// ---- CNC Beckhoff/6 BlockSearch/ReadBsBlockNumber.TcPOU
FUNCTION_BLOCK ReadBsBlockNumber
VAR_INPUT
	nIdxGrp: UDINT;
	bStart: BOOL;
	pDest: POINTER TO DINT;
END_VAR
VAR_OUTPUT
	Busy: BOOL;
	bErr: BOOL;
END_VAR
VAR
	fbRead: ADSREAD;
	bStarted: BOOL;
END_VAR

IF bStarted = FALSE THEN
   IF bStart = TRUE THEN
      bStarted := TRUE;
      bErr := FALSE;
      Busy := TRUE;
   END_IF
END_IF

IF bStarted THEN
   (* raising edge of Timer triggers read request *)
   fbRead( NetID := '', Port := 553, IdxGrp := nIdxGrp, IdxOffs := 16#00000077,
         LEN := 4, DestAddr := pDest, READ := bStarted, TMOUT := T#1s);
   IF NOT fbRead.Busy THEN
      (* There was an error in the execution of the read request *)
      IF fbRead.Err THEN
         bErr := TRUE;
      END_IF
      fbRead(READ := FALSE);    (* reset because of edge detection in FB ADSREAD *)
      bStarted := FALSE;
      Busy := FALSE;
   END_IF
END_IF

END_FUNCTION_BLOCK

// ---- CNC Beckhoff/6 BlockSearch/WriteBsBlockCount.TcPOU
FUNCTION_BLOCK WriteBsBlockCount
VAR_INPUT
	nIdxGrp: UDINT;
	bStart: BOOL;
	nBlockCount: DINT;
END_VAR
VAR_OUTPUT
	Busy: BOOL;
	bErr: BOOL;
END_VAR
VAR
	fbWrite: ADSWRITE;
	bStarted: BOOL;
END_VAR

IF bStarted = FALSE THEN
   IF bStart = TRUE THEN
      bStarted := TRUE;
      bErr := FALSE;
      Busy := TRUE;
   END_IF
END_IF

IF bStarted THEN
   (* raising edge of Timer triggers write request *)
   fbWrite( NetID := '', Port := 553, IdxGrp := nIdxGrp, IdxOffs := 16#0000005E,
         LEN := 4, SrcAddr := ADR(nBlockCount), WRITE := bStarted, TMOUT := T#1s);
   IF NOT fbWrite.Busy THEN
      (* There was an error in the execution of the write request *)
      IF fbWrite.Err THEN
         bErr := TRUE;
      END_IF
      fbWrite(WRITE := FALSE);    (* reset because of edge detection in FB ADSWRITE *)
      bStarted := FALSE;
      Busy := FALSE;
   END_IF
END_IF

END_FUNCTION_BLOCK

// ---- CNC Beckhoff/6 BlockSearch/ReadBlockCount.TcPOU
FUNCTION_BLOCK ReadBlockCount
VAR_INPUT
	nIdxGrp: UDINT;
	bStart: BOOL;
	pDest: POINTER TO DINT;
END_VAR
VAR_OUTPUT
	Busy: BOOL;
	bErr: BOOL;
END_VAR
VAR
	fbRead: ADSREAD;
	bStarted: BOOL;
END_VAR

IF bStarted = FALSE THEN
   IF bStart = TRUE THEN
      bStarted := TRUE;
      bErr := FALSE;
      Busy := TRUE;
   END_IF
END_IF

IF bStarted THEN
   (* raising edge of Timer triggers read request *)
   fbRead( NetID := '', Port := 553, IdxGrp := nIdxGrp, IdxOffs := 16#0000000D,
         LEN := 4, DestAddr := pDest, READ := bStarted, TMOUT := T#1s);
   IF NOT fbRead.Busy THEN
      (* There was an error in the execution of the read request *)
      IF fbRead.Err THEN
         bErr := TRUE;
      END_IF
      fbRead(READ := FALSE);    (* reset because of edge detection in FB ADSREAD *)
      bStarted := FALSE;
      Busy := FALSE;
   END_IF
END_IF

END_FUNCTION_BLOCK

// ---- CNC Beckhoff/6 BlockSearch/ReadBsBlockCount.TcPOU
FUNCTION_BLOCK ReadBsBlockCount
VAR_INPUT
	nIdxGrp: UDINT;
	bStart: BOOL;
	pDest: POINTER TO DINT;
END_VAR
VAR_OUTPUT
	Busy: BOOL;
	bErr: BOOL;
END_VAR
VAR
	fbRead: ADSREAD;
	bStarted: BOOL;
END_VAR

IF bStarted = FALSE THEN
   IF bStart = TRUE THEN
      bStarted := TRUE;
      bErr := FALSE;
      Busy := TRUE;
   END_IF
END_IF

IF bStarted THEN
   (* raising edge of Timer triggers read request *)
   fbRead( NetID := '', Port := 553, IdxGrp := nIdxGrp, IdxOffs := 16#00000076,
         LEN := 4, DestAddr := pDest, READ := bStarted, TMOUT := T#1s);
   IF NOT fbRead.Busy THEN
      (* There was an error in the execution of the read request *)
      IF fbRead.Err THEN
         bErr := TRUE;
      END_IF
      fbRead(READ := FALSE);    (* reset because of edge detection in FB ADSREAD *)
      bStarted := FALSE;
      Busy := FALSE;
   END_IF
END_IF

END_FUNCTION_BLOCK

// ---- CNC Beckhoff/6 BlockSearch/WriteBsPass.TcPOU
FUNCTION_BLOCK WriteBsPass
VAR_INPUT
	nIdxGrp: UDINT;
	bStart: BOOL;
	nPass: DINT;
END_VAR
VAR_OUTPUT
	Busy: BOOL;
	bErr: BOOL;
END_VAR
VAR
	fbWrite: ADSWRITE;
	bStarted: BOOL;
END_VAR

IF bStarted = FALSE THEN
   IF bStart = TRUE THEN
      bStarted := TRUE;
      bErr := FALSE;
      Busy := TRUE;
   END_IF
END_IF

IF bStarted THEN
   (* raising edge of Timer triggers write request *)
   fbWrite( NetID := '', Port := 553, IdxGrp := nIdxGrp, IdxOffs := 16#00000060,
         LEN := 4, SrcAddr := ADR(nPass), WRITE := bStarted, TMOUT := T#1s);
   IF NOT fbWrite.Busy THEN
      (* There was an error in the execution of the write request *)
      IF fbWrite.Err THEN
         bErr := TRUE;
      END_IF
      fbWrite(WRITE := FALSE);    (* reset because of edge detection in FB ADSWRITE *)
      bStarted := FALSE;
      Busy := FALSE;
   END_IF
END_IF

END_FUNCTION_BLOCK

// ---- CNC Beckhoff/6 BlockSearch/ReadBsPass.TcPOU
FUNCTION_BLOCK ReadBsPass
VAR_INPUT
	nIdxGrp: UDINT;
	bStart: BOOL;
	pDest: POINTER TO DINT;
END_VAR
VAR_OUTPUT
	Busy: BOOL;
	bErr: BOOL;
END_VAR
VAR
	fbRead: ADSREAD;
	bStarted: BOOL;
END_VAR

IF bStarted = FALSE THEN
   IF bStart = TRUE THEN
      bStarted := TRUE;
      bErr := FALSE;
      Busy := TRUE;
   END_IF
END_IF

IF bStarted THEN
   (* raising edge of Timer triggers read request *)
   fbRead( NetID := '', Port := 553, IdxGrp := nIdxGrp, IdxOffs := 16#00000078,
         LEN := 4, DestAddr := pDest, READ := bStarted, TMOUT := T#1s);
   IF NOT fbRead.Busy THEN
      (* There was an error in the execution of the read request *)
      IF fbRead.Err THEN
         bErr := TRUE;
      END_IF
      fbRead(READ := FALSE);    (* reset because of edge detection in FB ADSREAD *)
      bStarted := FALSE;
      Busy := FALSE;
   END_IF
END_IF

END_FUNCTION_BLOCK

// ---- CNC Beckhoff/2 OperationMode/ModeManual/HLI3_ManualModeHandler.TcPOU
FUNCTION_BLOCK HLI3_ManualModeHandler
VAR_INPUT
	stManualModeParameter: ST_ManualModeParameter;
	stManualModeControlElements: ST_ManualModeControlElements;
	bReset: BOOL;
END_VAR
VAR_OUTPUT
	bInManualMode: BOOL;
	arrAxisInG201: ARRAY[0..HLI_KEY_MAXIDX] OF UINT;
	bBusy: BOOL;
	bError: BOOL;
	nErrorId: INT;
END_VAR
VAR_IN_OUT
	stManualModeControlElementState: ST_ManualModeControlElementState;
END_VAR
VAR
	nState: INT;
	pString: POINTER TO STRING;
	pUnit: POINTER TO MC_CONTROL_MCM_MODE_STATE_UNIT;
	pCommand: POINTER TO HLI_PROC_TRANS_TO_MODE_STATE;
	pKey: POINTER TO MC_CONTROL_HB_KEY_UNIT;
	pIncr: POINTER TO MC_CONTROL_HB_TIP_PARAM_UNIT;
	stManualModeParameterOld: ST_ManualModeParameter;
	incOld: UINT;
	nManualTypOld: UINT;
	i: INT;
	bManual: BOOL;
	/// FBs for manual mode 
	ManualActivation: HLI3_ManualActivation;
	ManualExecution: ARRAY[0..HLI_KEY_MAXIDX] OF HLI3_ManualExecution;
	ManualExecutionRapidMode: ARRAY[0..HLI_KEY_MAXIDX] OF HLI3_ManualExecutionRapidMode;
	ActChannelModeOld: UDINT;
	TON_TimeOut: TON;
	nChan: INT;
	j: INT;
	strInitParameterOld: STRING;
	bInJoystickMode: BOOL;
	nHliAxisIdx: INT;
	nControlUnit: INT;
	arrAxisInJoystickMode: ARRAY[0..HLI_KEY_MAXIDX] OF UINT;
	n: INT;
	bInit: BOOL;
END_VAR
VAR CONSTANT
	ErrID_1: INT := 1;
END_VAR

(* ========================================================= 	*)
(*     FB: HLI3_ManualModeHandler                           	*)
(* --------------------------------------------------------- 	*)
(*   Desc: Switch to Manual Mode and parametrize             	*)
(*   Author: MK / TV  /MiB                                      *)
(*   Date: 18.07.2002                                        	*)
(*   Last: 18.11.2015                                        	*)
(*   Rev.: 6.4	                                              	*)
(* ========================================================= 	*)

nChan := stManualModeParameter.stChannelParameter.nChanIdx;
IF (NOT HLI3_CheckChannelValid(nChannel := nChan) OR nChan = -1 )  THEN
	RETURN;
END_IF

IF NOT bInit THEN  
	gpCh[nChan]^.hb_mc_control.activation.enable_w := TRUE;
	FOR j := 0 TO HLI_HW_MAXIDX DO
		gpCh[nChan]^.hb_mc_control.handwheel_incs[j].enable_w  := TRUE;
	END_FOR
	bInit := TRUE;
END_IF	

IF 	CNCSystem.Channel[nChan].ActMode <> HLI_IMCM_MANUAL_MODE AND
	CNCSystem.Channel[nChan].ActMode <> HLI_IMCM_AUTOMATIC_MODE   AND
	CNCSystem.Channel[nChan].ActMode <> HLI_IMCM_MDI_MODE THEN
		strInitParameterOld := '';
		bBusy := FALSE;
		nState := 0;
	RETURN; (* A b b r u c h *)
ELSE
	bManual := TRUE;
END_IF

IF  CNCSystem.Channel[nChan].ActMode <> HLI_IMCM_MANUAL_MODE THEN
	strInitParameterOld := '';
END_IF

(* Clear all request from the HMI *)
IF gpCh[nChan]^.hb_mc_control.key[0].request_semaphor_rw THEN
	gpCh[nChan]^.hb_mc_control.key[0].request_semaphor_rw := FALSE;
END_IF

IF gpCh[nChan]^.hb_mc_control.activation.request_semaphor_rw THEN
	gpCh[nChan]^.hb_mc_control.activation.request_semaphor_rw := FALSE;
END_IF

IF gpCh[nChan]^.hb_mc_control.tip_parameter.request_semaphor_rw THEN
	gpCh[nChan]^.hb_mc_control.tip_parameter.request_semaphor_rw := FALSE;
END_IF

IF gpCh[nChan]^.hb_mc_control.jog_parameter.request_semaphor_rw THEN
	gpCh[nChan]^.hb_mc_control.jog_parameter.request_semaphor_rw := FALSE;
END_IF

bBusy := TRUE;

IF bReset THEN		
	bError := FALSE;
	nErrorID := 0;
	bInManualMode := FALSE;
END_IF


IF stManualModeParameter.stChannelParameter.eManualType = E_CNC_ManualType.JoystickMode THEN

	bInJoystickMode := TRUE;
	
	arrAxisInJoystickMode := HLI3_LogicalAxisInManualMode(nCHan);
	
	PRG_AnalogJoystick(	nLogAxisNr:= stManualModeParameter.stAxisParameter.stControlUnit[0].nLogAxisNr,
								Analog_Value:= stManualModeControlElements.stControlJoystickValue[0],
								AnalogValueMin:= stManualModeParameter.stJoystickParameter.AnalogValueMin,
								AnalogValueMax:= stManualModeParameter.stJoystickParameter.AnalogValueMax,
								AnalogValueZeroDeadBand:= stManualModeParameter.stJoystickParameter.AnalogValueZeroDeadBand,
								bKeyPos:= stManualModeControlElements.stControlKeys[0].bKeyPos,
								bKeyNeg:= stManualModeControlElements.stControlKeys[0].bKeyNeg);

	PRG_AnalogJoystick(	nLogAxisNr:= stManualModeParameter.stAxisParameter.stControlUnit[1].nLogAxisNr,
								Analog_Value:= stManualModeControlElements.stControlJoystickValue[1],
								AnalogValueMin:= stManualModeParameter.stJoystickParameter.AnalogValueMin,
								AnalogValueMax:= stManualModeParameter.stJoystickParameter.AnalogValueMax,
								AnalogValueZeroDeadBand:= stManualModeParameter.stJoystickParameter.AnalogValueZeroDeadBand,
								bKeyPos:= stManualModeControlElements.stControlKeys[1].bKeyPos,
								bKeyNeg:= stManualModeControlElements.stControlKeys[1].bKeyNeg);

	PRG_AnalogJoystick(	nLogAxisNr:= stManualModeParameter.stAxisParameter.stControlUnit[2].nLogAxisNr,
								Analog_Value:= stManualModeControlElements.stControlJoystickValue[2],
								AnalogValueMin:= stManualModeParameter.stJoystickParameter.AnalogValueMin,
								AnalogValueMax:= stManualModeParameter.stJoystickParameter.AnalogValueMax,
								AnalogValueZeroDeadBand:= stManualModeParameter.stJoystickParameter.AnalogValueZeroDeadBand,
								bKeyPos:= stManualModeControlElements.stControlKeys[2].bKeyPos,
								bKeyNeg:= stManualModeControlElements.stControlKeys[2].bKeyNeg);

	PRG_AnalogJoystick(	nLogAxisNr:= stManualModeParameter.stAxisParameter.stControlUnit[3].nLogAxisNr,
								Analog_Value:= stManualModeControlElements.stControlJoystickValue[3],
								AnalogValueMin:= stManualModeParameter.stJoystickParameter.AnalogValueMin,
								AnalogValueMax:= stManualModeParameter.stJoystickParameter.AnalogValueMax,
								AnalogValueZeroDeadBand:= stManualModeParameter.stJoystickParameter.AnalogValueZeroDeadBand,
								bKeyPos:= stManualModeControlElements.stControlKeys[3].bKeyPos,
								bKeyNeg:= stManualModeControlElements.stControlKeys[3].bKeyNeg);

	PRG_AnalogJoystick(	nLogAxisNr:= stManualModeParameter.stAxisParameter.stControlUnit[4].nLogAxisNr,
								Analog_Value:= stManualModeControlElements.stControlJoystickValue[4],
								AnalogValueMin:= stManualModeParameter.stJoystickParameter.AnalogValueMin,
								AnalogValueMax:= stManualModeParameter.stJoystickParameter.AnalogValueMax,
								AnalogValueZeroDeadBand:= stManualModeParameter.stJoystickParameter.AnalogValueZeroDeadBand,
								bKeyPos:= stManualModeControlElements.stControlKeys[4].bKeyPos,
								bKeyNeg:= stManualModeControlElements.stControlKeys[4].bKeyNeg);

ELSE
	(* Achsoverride wieder auf 100 % setzen *)
	IF bInJoystickMode THEN 
		nHliAxisIdx := -1;
		FOR j := 0 TO UINT_TO_INT(SIZEOF(arrAxisInJoystickMode)) DO
			FOR i := 0 TO UDINT_TO_INT(gNrAx-1) DO
				IF (gpAX[i]^.head.log_ax_nr_r = arrAxisInJoystickMode[j]) THEN
					nHliAxisIdx := i;	
					IF (nHliAxisIdx <> -1) THEN 
						HLI3_SetAxisOverride(nHliAxisIdx := nHliAxisIdx, nOverride := 1000);
						nHliAxisIdx := -1;
						arrAxisInJoystickMode[j] := 0;
					END_IF								
				END_IF
			END_FOR			
		END_FOR
		bInJoystickMode := FALSE;
	END_IF
END_IF

(******** Parallelinterpolation mit G201 *************************************)
IF CNCSystem.Channel[nChan].ActMode = HLI_IMCM_AUTOMATIC_MODE OR CNCSystem.Channel[nChan].ActMode = HLI_IMCM_MDI_MODE THEN
	arrAxisInG201 := HLI3_LogicalAxisInManualMode(nCHan);
	FOR j := 0 TO HLI_KEY_MAXIDX DO
		stManualModeParameter.stAxisParameter.stControlUnit[j].nLogAxisNr := arrAxisInG201[j];
	END_FOR
ELSE
	FOR j := 0 TO HLI_KEY_MAXIDX DO
		arrAxisInG201[j] := 0;
	END_FOR
END_IF
(* **************************************************************************** *)

IF NOT gpCh[nChan]^.bahn_state.g201_active_r THEN
	IF CNCSystem.Channel[nChan].ActMode = HLI_IMCM_AUTOMATIC_MODE OR CNCSystem.Channel[nChan].ActMode = HLI_IMCM_MDI_MODE THEN
		nState := 0; 
	END_IF
END_IF

CASE nState OF


	0: (* IDLE *)
		bBusy := FALSE;
		bInManualMode := FALSE;


		IF (CNCSystem.Channel[nChan].ActMode = HLI_IMCM_MANUAL_MODE AND
    		stManualModeParameter.stChannelParameter.eManualType <> E_CNC_ManualType.NoManualMode AND
    		CNCSystem.Channel[nChan].ActState = HLI_IMCM_PROCESS_ACTIVE) OR  (* Manual Mode *)
   			((arrAxisinG201[0] <> 0)    (* mindestens eine Achse in G201 *) AND
    		((CNCSystem.Channel[nChan].ActState = HLI_IMCM_PROCESS_ACTIVE) OR
     		(CNCSystem.Channel[nChan].ActState = HLI_IMCM_PROCESS_HOLD))) (* Channel is active *)
		THEN			
			bError 		:= FALSE;
			nErrorID 	:= 0;

			stManualModeParameterOld     := stManualModeParameter;
			ActChannelModeOld   		:= cncsystem.Channel[nChan].ActMode;			
			i:= 0;
			nState := 10;

		END_IF

	10:		// Restore Manual State										
			FOR j := 0 TO HLI_KEY_MAXIDX DO
				IF (stManualModeControlElementState.stKeyUnit[j].nChan = nChan) THEN
					stManualModeControlElementState.stKeyUnit[j].nChan := -1;
					stManualModeControlElementState.stKeyUnit[j].nLogAxisId := 0;
					stManualModeControlElementState.stKeyUnit[j].nInputParameterIdx := -1;
				END_IF													
			END_FOR
			
			FOR j := 0 TO HLI_HW_MAXIDX DO
				IF (stManualModeControlElementState.stHWUnit[j].nChan = nChan) THEN
					stManualModeControlElementState.stHWUnit[j].nChan := -1;
					stManualModeControlElementState.stHWUnit[j].nLogAxisId := 0;
					stManualModeControlElementState.stHWUnit[j].nInputParameterIdx := -1;
				END_IF													
			END_FOR
			(*
			FOR j := 0 TO HLI_CH_AX_MAXIDX DO
				IF gpCh[nChan]^.bahn_state.coord_r[j].hb_display_r.control_element <> 0 THEN
					IF gpCh[nChan]^.bahn_state.coord_r[j].hb_display_r.operation_mode = 1 THEN  
						stManualModeControlElementState.stHWUnit[gpCh[nChan]^.bahn_state.coord_r[j].hb_display_r.control_element-1].nLogAxisId := gpCh[nChan]^.bahn_state.coord_r[j].log_achs_nr_r;
 						stManualModeControlElementState.stHWUnit[gpCh[nChan]^.bahn_state.coord_r[j].hb_display_r.control_element-1].nChan := nChan;
					ELSE
						stManualModeControlElementState.stKeyUnit[gpCh[nChan]^.bahn_state.coord_r[j].hb_display_r.control_element-1].nLogAxisId := gpCh[nChan]^.bahn_state.coord_r[j].log_achs_nr_r;
 						stManualModeControlElementState.stKeyUnit[gpCh[nChan]^.bahn_state.coord_r[j].hb_display_r.control_element-1].nChan := nChan;
					END_IF
				END_IF 
			END_FOR
*)	
			n:= 0;		
			nState := 20;						
			
20: 	// Deactivation 
		IF (n <= HLI_CH_AX_MAXIDX) THEN
			IF gpCh[nChan]^.bahn_state.coord_r[n].hb_display_r.control_element <> 0 THEN 
				IF NOT gpCh[nChan]^.hb_mc_control.activation.command_semaphor_rw THEN		
						gpCh[nChan]^.hb_mc_control.activation.command_w.log_achs_nr := gpCh[nChan]^.bahn_state.coord_r[n].log_achs_nr_r;
						gpCh[nChan]^.hb_mc_control.activation.command_w.control_element := 0;
						gpCh[nChan]^.hb_mc_control.activation.command_w.operation_mode := 0;
						
						IF (gpCh[nChan]^.bahn_state.coord_r[n].hb_display_r.operation_mode = 1) THEN
							stManualModeControlElementState.stHWUnit[gpCh[nChan]^.bahn_state.coord_r[n].hb_display_r.control_element-1].nChan := -1;
							stManualModeControlElementState.stHWUnit[gpCh[nChan]^.bahn_state.coord_r[n].hb_display_r.control_element-1].nLogAxisId :=0;
							stManualModeControlElementState.stHWUnit[gpCh[nChan]^.bahn_state.coord_r[n].hb_display_r.control_element-1].nInputParameterIdx := -1;	
						ELSE
							stManualModeControlElementState.stKeyUnit[gpCh[nChan]^.bahn_state.coord_r[n].hb_display_r.control_element-1].nChan := -1;
							stManualModeControlElementState.stKeyUnit[gpCh[nChan]^.bahn_state.coord_r[n].hb_display_r.control_element-1].nLogAxisId :=0;
							stManualModeControlElementState.stKeyUnit[gpCh[nChan]^.bahn_state.coord_r[n].hb_display_r.control_element-1].nInputParameterIdx := -1;						
						END_IF
						gpCh[nChan]^.hb_mc_control.activation.command_semaphor_rw := TRUE;
						nState := 21;					
				END_IF
			ELSE
				n := n + 1;
			END_IF				
		END_IF

		IF n >HLI_CH_AX_MAXIDX THEN
			nState := 26;
		END_IF
21: 
		IF 	NOT gpCh[nChan]^.hb_mc_control.activation.command_semaphor_rw THEN						
			n := n+1;
			nState := 20;
		END_IF
		
		IF n > HLI_CH_AX_MAXIDX THEN
			nState := 26;
		END_IF			
			 					
		(* Activation of an manual mode string, eg. TRAFO ON or ECS ON *)
26:     IF 	(stManualModeParameter.stChannelParameter.strInitParameter  <> '' AND
			stManualModeParameter.stChannelParameter.strInitParameter <> strInitParameterOld AND
			CNCSystem.Channel[nChan].ActMode = HLI_IMCM_MANUAL_MODE) THEN
			gpCh[nCHan]^.channel_mc_control.mode_and_state.command_w.to_mode := HLI_IMCM_MANUAL_MODE ;
			gpCh[nCHan]^.channel_mc_control.mode_and_state.command_w.to_state := HLI_IMCM_PROCESS_SELECTED;
			gpCh[nCHan]^.channel_mc_control.mode_and_state.command_w.channel_number := INT_TO_UDINT(nChan+1);
			pString := ADR(gpCh[nCHan]^.channel_mc_control.mode_and_state.command_w.parameter);
			pString^ := '';
			gpCh[nChan]^.channel_mc_control.mode_and_state.command_semaphor_rw := TRUE;
			TON_TimeOut(in:= FALSE);
			nState := 27;
		ELSE
			i := 0;
			nState := 30;
		END_IF


27:		IF (gpCh[nCHan]^.channel_mc_control.mode_and_state.command_semaphor_rw = FALSE) AND 
			CNCSystem.Channel[nChan].ActState = HLI_IMCM_PROCESS_SELECTED 
		THEN
			gpCh[nCHan]^.channel_mc_control.mode_and_state.command_w.to_mode := HLI_IMCM_MANUAL_MODE ;
			gpCh[nCHan]^.channel_mc_control.mode_and_state.command_w.to_state := HLI_IMCM_PROCESS_ACTIVE;
			gpCh[nCHan]^.channel_mc_control.mode_and_state.command_w.channel_number := INT_TO_UDINT(nChan+1);
			pString := ADR(gpCh[nCHan]^.channel_mc_control.mode_and_state.command_w.parameter);
			pString^ := stManualModeParameter.stChannelParameter.strInitParameter;
			gpCh[nCHan]^.channel_mc_control.mode_and_state.command_semaphor_rw := TRUE;		
			TON_TimeOut(in:= FALSE);		
			nState := 28;
		END_IF

		TON_TimeOut(in:=TRUE, PT:=T#5s);
		IF TON_TimeOut.Q THEN
			nState := 99;
		END_IF

28:		IF (gpCh[nCHan]^.channel_mc_control.mode_and_state.command_semaphor_rw = FALSE)  AND
			CNCSystem.Channel[nChan].ActState = HLI_IMCM_PROCESS_ACTIVE 
			THEN														
				strInitParameterOld := stManualModeParameter.stChannelParameter.strInitParameter;
				ManualActivation(bExecute := FALSE,stManualModeControlElementState:= stManualModeControlElementState);
				i := 0;
				IF (gpCh[nChan]^.bahn_state.g200_active_r) THEN	
					nState := 30;
				END_IF
						
		END_IF	

		// Abbruch wenn die Betriebsart gewechselt wird 
		IF (CNCSystem.Channel[nChan].ActMode <> HLI_IMCM_MANUAL_MODE) THEN
			nState := 0;
		END_IF	
	
30: 	(* --- activate KeyControlUnits --- *)														
		ManualActivation(bExecute := TRUE,
									nChan 			 := nChan,
									eManualType 	 := stManualModeParameter.stChannelParameter.eManualType,									
									stManualModeControlElementState:= stManualModeControlElementState,
									nInputParameterIdx := i,
									nHBA_Res 		 := stManualModeParameter.stChannelParameter.nHandwheelResolution,
									Inc 		     := stManualModeParameter.stChannelParameter.nInc,
									Speed 			 := stManualModeParameter.stAxisParameter.stControlUnit[i].nSpeed, // geändert alt nControlUnit
									nLogAxisNr 		 := stManualModeParameter.stAxisParameter.stControlUnit[i].nLogAxisNr); // geändert alt nControlUnit
		nState := 35;				
															
35: 	(* waiting for acknowledge *)
		ManualActivation(bExecute := FALSE, stManualModeControlElementState:= stManualModeControlElementState);
		
		IF ManualActivation.bBusy = FALSE THEN
			IF ManualActivation.bError THEN
				nErrorId := ErrID_1;
				nState := 99;
			ELSE
				IF stManualModeParameter.stAxisParameter.stControlUnit[i+1].nLogAxisNr = 0 THEN
					i:=-1; (* reset the array counter *)				
					nState := 40;
				ELSE
					ManualActivation(bExecute := FALSE, stManualModeControlElementState:= stManualModeControlElementState);
					nState := 30;
					i:= i+1;
				END_IF
			END_IF
		END_IF

40: 	(* endlich Handbetrieb *)
		bInManualMode := TRUE;
		
		IF (stManualModeParameter.stChannelParameter.eManualType <> E_CNC_ManualType.Handwheel) THEN
			FOR j := 0 TO HLI_KEY_MAXIDX DO
				IF stManualModeControlElementState.stKeyUnit[j].nChan = nChan AND stManualModeControlElementState.stKeyUnit[j].nLogAxisId <> 0 THEN				
					ManualExecution[j](	nChan := nChan,
									nKeyControlUnit := j,
									bKeyPos := stManualModeControlElements.stControlKeys[stManualModeControlElementState.stKeyUnit[j].nInputParameterIdx].bKeyPos,					// geändert 	nControlUnit
									bKeyNeg := stManualModeControlElements.stControlKeys[stManualModeControlElementState.stKeyUnit[j].nInputParameterIdx].bKeyNeg); (* no timeouts *)
									
					ManualExecutionRapidMode[j](nChan := nChan,
									nKeyControlUnit := j,
									bExecute := stManualModeControlElements.stControlKeys[stManualModeControlElementState.stKeyUnit[j].nInputParameterIdx].bKeyRapid); (* no timeouts *)
				END_IF
			END_FOR			
		ELSE				
			(* Handradincremente werden immer vom ersten Kanal entgegen genommen*)
			FOR j := 0 TO HLI_HW_MAXIDX DO
				IF (stManualModeControlElementState.stHWUnit[j].nChan = nChan AND stManualModeControlElementState.stHWUnit[j].nLogAxisId <>  0)  THEN 
					gpCh[0]^.hb_mc_control.handwheel_incs[j].command_w := stManualModeControlElements.nHandwheelInc[stManualModeControlElementState.stHWUnit[j].nInputParameterIdx];
				END_IF			
			END_FOR
		END_IF

		(* end of manual mode *)
		 IF (bManual = FALSE) OR                                                                                                             
         	MEMCMP(ADR(stManualModeParameter),ADR(stManualModeParameterOld),SIZEOF(stManualModeParameter)-SIZEOF(stManualModeParameter.stChannelParameter.strInitParameter))<>0 OR                                                      
            stManualModeParameter.stChannelParameter.strInitParameter <> stManualModeParameterOld.stChannelParameter.strInitParameter OR                                                          
            cncsystem.Channel[nChan].ActMode <> ActChannelModeOld OR                                       
            (CNCSystem.Channel[nChan].ActMode =  HLI_IMCM_MANUAL_MODE AND CNCSystem.Channel[nChan].ActState <> HLI_IMCM_PROCESS_ACTIVE) OR                                                   
            stManualModeParameter.stChannelParameter.eManualType = E_CNC_ManualType.NoManualMode
            THEN
		
				FOR j := 0 TO HLI_KEY_MAXIDX DO
					IF stManualModeControlElementState.stKeyUnit[j].nChan = nChan THEN
						ManualExecution[j](nChan := nChan,	nKeyControlUnit := j, bKeyPos := FALSE, bKeyNeg := FALSE); (* no timeouts *)		
					END_IF		
				END_FOR
						
				i:=1 (* resets the counter for the following deactivation *);			

				stManualModeParameterOld 	:= stManualModeParameter;
	
				IF cncsystem.Channel[nChan].ActMode <> ActChannelModeOld OR stManualModeParameter.stChannelParameter.eManualType = E_CNC_ManualType.NoManualMode THEN
					ActChannelModeOld := cncsystem.Channel[nChan].ActMode;			
					nState := 0;
				ELSE
					nState := 0; (* evt. wird hier auch eine Verzoegerungszeit benötigt,
										  Fehler 150054 dann nState = 0 *)
					bInManualMode := FALSE;
				END_IF
		END_IF

99: 	(* error handling *)	
		bBusy := FALSE;
		bError := TRUE;
		
		(* end of manual mode *)
			IF NOT gpCh[nCHan]^.channel_mc_control.mode_and_state.command_semaphor_rw AND 
			CNCSystem.Channel[nChan].ActState <>  HLI_IMCM_PROCESS_ERROR
			THEN;
				gpCh[nCHan]^.channel_mc_control.mode_and_state.command_w.to_mode := HLI_IMCM_MANUAL_MODE ;
				gpCh[nCHan]^.channel_mc_control.mode_and_state.command_w.to_state := HLI_IMCM_PROCESS_ERROR;
				gpCh[nCHan]^.channel_mc_control.mode_and_state.command_w.channel_number := INT_TO_UDINT(nChan+1);			
				gpCh[nCHan]^.channel_mc_control.mode_and_state.command_semaphor_rw := TRUE;	
			END_IF
			nState := 0;
		
		(* end of manual mode *)
		IF bManual = FALSE THEN
			bBusy := FALSE;
			nState := 0;
		END_IF

END_CASE

END_FUNCTION_BLOCK

// ---- CNC Beckhoff/2 OperationMode/ModeManual/HLI3_ManualActivation.TcPOU
FUNCTION_BLOCK HLI3_ManualActivation
VAR_INPUT
	bExecute: BOOL;
	/// Number of channel 
	nChan: INT;
	eManualType: E_CNC_ManualType;
	/// Increments -> 0 activates Tip mode 
	Inc: UDINT;
	/// Aufloesung des Achsverfahrwegs bei einer Handradumdrehung Einheit: 0.1um / Handradumdrehung
	nHBA_Res: DINT;
	Speed: UDINT;
	/// axis nr 
	nLogAxisNr: UINT;
	nInputParameterIdx: INT;
END_VAR
VAR_OUTPUT
	bError: BOOL;
	bBusy: BOOL;
END_VAR
VAR_IN_OUT
	stManualModeControlElementState: ST_ManualModeControlElementState;
END_VAR
VAR
	fbRtrigExec: R_TRIG;
	nState: INT;
	pActivation: POINTER TO MC_CONTROL_HB_ACTIVATION_UNIT;
	pJogParameter: POINTER TO MC_CONTROL_HB_JOG_PARAM_UNIT;
	pTipParameter: POINTER TO MC_CONTROL_HB_TIP_PARAM_UNIT;
	pHBHRParameter: POINTER TO MC_CONTROL_HB_HR_PARAM_UNIT;
	j: INT;
	bFreeControlElementFound: BOOL;
END_VAR

(* ========================================================= *)
(*    FUN: HLI_ManualActivation                       		 *)
(* --------------------------------------------------------- *)
(*   Desc:                                                   *)
(*   Author: CL TV MiB                                       *)
(*   Date: 18.11.2005                                        *)
(*   Last: 25.02.2015                                       *)
(*   Rev.: 6.0                                              *)
(* ========================================================= *)

IF NOT HLI3_CheckChannelValid(nChannel := nChan) OR nLogAxisNr = 0 THEN
	RETURN;
END_IF


fbRtrigExec(clk := bExecute);
IF fbRtrigExec.Q THEN
	bBusy := TRUE;
	bError := FALSE;
	nState := 10;
END_IF

CASE nState OF

	0: (* IDLE *)
		bBusy := FALSE;

	10:
		CASE eManualType OF
			E_CNC_ManualType.NoManualMode: 
				nState := 100;

			E_CNC_ManualType.Handwheel:
				nState := 30;

			E_CNC_ManualType.TippMode:
				nState := 40;

			E_CNC_ManualType.JogMode:
				nState := 50;

			E_CNC_ManualType.JoystickMode:
				nState := 40;

			E_CNC_ManualType.DigitalJoystick: 
				nState := 40;

		END_CASE

	30:(* Setze Handrad Parameter *)
		pHBHRParameter := ADR(gpCh[nChan]^.hb_mc_control.hr_parameter);
		IF NOT pHBHRParameter^.command_semaphor_rw THEN
			pHBHRParameter^.enable_w := TRUE;
			pHBHRParameter^.command_w.resolution  := nHBA_Res;
			pHBHRParameter^.command_w.log_achs_nr := nLogAxisNr;
			pHBHRParameter^.command_semaphor_rw := TRUE;
			nState := 100;
		END_IF

	40: (* Setze Parameter für den Tippbetrieb *)
		pTipParameter := ADR(gpCh[nChan]^.hb_mc_control.tip_parameter);
		IF NOT pTipParameter^.command_semaphor_rw THEN
			pTipParameter^.enable_w := TRUE;
			pTipParameter^.command_w.log_achs_nr := nLogAxisNr;
			pTipParameter^.command_w.speed       := Speed;
			pTipParameter^.command_semaphor_rw := TRUE;
			nState := 100;
		END_IF

	50: (* Setze Parameter für den Jogbetrieb *)
		pJogParameter := ADR(gpCh[nChan]^.hb_mc_control.jog_parameter);
		IF NOT pJogParameter^.command_semaphor_rw THEN
			pJogParameter^.enable_w := TRUE;
			pJogParameter^.command_w.log_achs_nr := nLogAxisNr;
			pJogParameter^.command_w.distance    := Inc;
			pJogParameter^.command_w.speed       := Speed;
			pJogParameter^.command_semaphor_rw := TRUE;
			nState := 100;
		END_IF		
		
	100: 	(* Aktivierung der Bedienelementen für den Handbetrieb  *)		
		
		pActivation := ADR(gpCh[nChan]^.hb_mc_control.activation);
		IF NOT pActivation^.command_semaphor_rw THEN 
			bFreeControlElementFound := FALSE;


			IF 	eManualType <> E_CNC_ManualType.Handwheel THEN 	
				FOR j := 0 TO HLI_KEY_MAXIDX DO
					IF stManualModeControlElementState.stKeyUnit[j].nLogAxisId = 0 THEN
							stManualModeControlElementState.stKeyUnit[j].nLogAxisId := nLogAxisNr;
							stManualModeControlElementState.stKeyUnit[j].nChan := nChan;
							stManualModeControlElementState.stKeyUnit[j].nInputParameterIdx := nInputParameterIdx;
							bFreeControlElementFound := TRUE;
						EXIT;
					END_IF 
				END_FOR
			ELSE
				FOR j := 0 TO HLI_HW_MAXIDX DO
					IF stManualModeControlElementState.stHWUnit[j].nLogAxisId = 0 THEN
							stManualModeControlElementState.stHWUnit[j].nLogAxisId := nLogAxisNr;
							stManualModeControlElementState.stHWUnit[j].nChan := nChan;
							stManualModeControlElementState.stHWUnit[j].nInputParameterIdx := nInputParameterIdx;
							bFreeControlElementFound := TRUE;
						EXIT;
					END_IF 
				END_FOR
			END_IF
							
			IF bFreeControlElementFound THEN
				pActivation^.enable_w := TRUE;
				pActivation^.command_w.log_achs_nr := nLogAxisNr;
				pActivation^.command_w.control_element := INT_TO_UINT(j+1);
		
		
				CASE eManualType OF
					E_CNC_ManualType.NoManualMode: 
						pActivation^.command_w.operation_mode := 0; 	(* 0 - No OP_Mode *)
		
					E_CNC_ManualType.Handwheel: 
						pActivation^.command_w.operation_mode := 1; 	(* 1 - Handwheel *)
		
					E_CNC_ManualType.TippMode: 
						pActivation^.command_w.operation_mode := 2; 	(* 2 - Tip Mode continous *)
		
					E_CNC_ManualType.JogMode: 
						pActivation^.command_w.operation_mode := 3; 	(* 3 - Jog Mode (incremental *)
		
					E_CNC_ManualType.JoystickMode: 
						pActivation^.command_w.operation_mode := 2; 	(* 2 - Tip Mode continous, auch für Analog Joystick *)
		
					E_CNC_ManualType.DigitalJoystick: 
						pActivation^.command_w.operation_mode := 2; 	(* 2 - Tip Mode continous, auch für Digital Joystick *)
		
				END_CASE
			
				pActivation^.command_semaphor_rw := TRUE;
				nState := 0;
			ELSE
				bError := TRUE;
				nState := 0;
			END_IF
		END_IF						
END_CASE

END_FUNCTION_BLOCK

// ---- CNC Beckhoff/2 OperationMode/ModeManual/HLI3_ManualExecution.TcPOU
FUNCTION_BLOCK HLI3_ManualExecution
VAR_INPUT
	nChan: INT;
	/// number of the HB_KeyControlUnit 
	nKeyControlUnit: INT;
	/// static signal 
	bKeyPos: BOOL;
	/// static signal 
	bKeyNeg: BOOL;
END_VAR
VAR
	Cmd_Dir: E_HLI_MM_KEYDirection;
	Act_Dir: E_HLI_MM_KEYDirection;
END_VAR

(* ========================================================= *)
(*    FUN: HLI_ManualExecution                    		 		 *)
(* --------------------------------------------------------- *)
(*   Desc:                                                   *)
(*   Author: CL / TV                                         *)
(*   Date: 24.07.2015                                       *)
(*   Rev.: 6.0                                               *)
(* ========================================================= *)

(* flank detection second axis*)
gpCh[nChan]^.hb_mc_control.key[nKeyControlUnit].enable_w := TRUE;

IF (NOT bKeyPos AND NOT bKeyNeg) OR (bKeyPos AND Act_Dir = KEY_DIR_NEGATIVE) OR (bKeyNeg AND Act_Dir = KEY_DIR_POSITIVE) THEN
	Cmd_Dir := KEY_DIR_NOT_PRESSED;
	IF NOT gpCh[nChan]^.hb_mc_control.key[nKeyControlUnit].command_semaphor_rw AND Cmd_dir <> Act_Dir THEN
		gpCh[nChan]^.hb_mc_control.key[nKeyControlUnit].command_w.log_key_nr := DINT_TO_UINT(nKeyControlUnit)+1;
		gpCh[nChan]^.hb_mc_control.key[nKeyControlUnit].command_w.direction := KEY_DIR_NOT_PRESSED;
		gpCh[nChan]^.hb_mc_control.key[nKeyControlUnit].command_semaphor_rw := TRUE;
		Act_Dir := KEY_DIR_NOT_PRESSED;
	END_IF	
END_IF


IF bKeyPos AND Act_Dir = KEY_DIR_NOT_PRESSED THEN
	Cmd_Dir := KEY_DIR_POSITIVE;
	IF NOT gpCh[nChan]^.hb_mc_control.key[nKeyControlUnit].command_semaphor_rw AND Cmd_dir <> Act_Dir THEN
		gpCh[nChan]^.hb_mc_control.key[nKeyControlUnit].command_w.log_key_nr := DINT_TO_UINT(nKeyControlUnit)+1;
		gpCh[nChan]^.hb_mc_control.key[nKeyControlUnit].command_w.direction := KEY_DIR_POSITIVE;
		gpCh[nChan]^.hb_mc_control.key[nKeyControlUnit].command_semaphor_rw := TRUE;
		Act_Dir := KEY_DIR_POSITIVE;
	END_IF	
END_IF

IF bKeyNeg AND Act_Dir = KEY_DIR_NOT_PRESSED  THEN
	Cmd_Dir := KEY_DIR_NEGATIVE;
	IF NOT gpCh[nChan]^.hb_mc_control.key[nKeyControlUnit].command_semaphor_rw AND Cmd_dir <> Act_Dir THEN
		gpCh[nChan]^.hb_mc_control.key[nKeyControlUnit].command_w.log_key_nr := DINT_TO_UINT(nKeyControlUnit)+1;
		gpCh[nChan]^.hb_mc_control.key[nKeyControlUnit].command_w.direction := KEY_DIR_NEGATIVE;
		gpCh[nChan]^.hb_mc_control.key[nKeyControlUnit].command_semaphor_rw := TRUE;
		Act_Dir := KEY_DIR_NEGATIVE;
	END_IF	
END_IF

END_FUNCTION_BLOCK

// ---- CNC Beckhoff/2 OperationMode/ModeManual/HLI3_ManualExecutionRapidMode.TcPOU
FUNCTION_BLOCK HLI3_ManualExecutionRapidMode
VAR_INPUT
	nChan: INT;
	/// number of the HB_KeyControlUnit 
	nKeyControlUnit: INT;
	/// static signal 
	bExecute: BOOL;
END_VAR
VAR
	pRapidKey: POINTER TO MC_CONTROL_HB_RAPID_KEY_UNIT;
	TONTimeOut: TON;
	fbRtrigExec: R_TRIG;
	fbFtrigExec: F_TRIG;
END_VAR

(* ========================================================= *)
(*    FUN: HLI_ManualExecution                               *)
(* --------------------------------------------------------- *)
(*   Desc:                                                   *)
(*   Author: TV                                              *)
(*   Date: 24.07.2015                                        *)
(*   Rev.: 6.0                                               *)
(* ========================================================= *)


IF nKeyControlUnit < 0 OR nKeyControlUnit > HLI_KEY_MAXIDX THEN
	RETURN;
END_IF;

pRapidKey := ADR(gpCh[nChan]^.hb_mc_control.rapid_key);
pRapidKey^.enable_w := TRUE;

IF NOT pRapidKey^.command_semaphor_rw THEN
	fbRtrigExec(clk := bExecute);
	fbFtrigExec(clk := bExecute);
END_IF

IF fbRtrigExec.Q THEN
	pRapidKey^.command_w.key_pressed := 1;
	pRapidKey^.command_w.log_key_nr := INT_TO_UINT(nKeyControlUnit)+1;
	pRapidKey^.command_semaphor_rw := TRUE;
END_IF


IF fbFtrigExec.Q THEN
	pRapidKey^.command_w.key_pressed := 0;
	pRapidKey^.command_w.log_key_nr := INT_TO_UINT(nKeyControlUnit)+1;
	pRapidKey^.command_semaphor_rw := TRUE;
END_IF

END_FUNCTION_BLOCK

// ---- CNC Beckhoff/2 OperationMode/ModeManual/HLI3_LogicalAxisInManualMode.TcPOU
FUNCTION HLI3_LogicalAxisInManualMode : ARRAY[0..HLI_KEY_MAXIDX] OF UINT
VAR_INPUT
	nChan: INT;
END_VAR
VAR
	i: INT;
	n: INT;
END_VAR

(* 		  If no axis is in manual mode it returns 0           		*)
(* Author: MiB/TV                                         			*)
(*   Date: 16.07.2007                                         		*)
(*   Last: 05.04.2016                                        		*)
(*   Rev.: 1.1                                                 		*)
(* ================================================================= *)

IF (NOT HLI3_CheckChannelValid(nChannel := nChan)) THEN
	RETURN;
END_IF

n:= 0;
FOR i := 0 TO HLI_CH_AX_MAXIDX DO
  	IF (gpCh[nChan]^.bahn_state.coord_r[i].hb_display_r.state <> 0) THEN
		HLI3_LogicalAxisInManualMode[n] := gpCh[nChan]^.bahn_state.coord_r[i].log_achs_nr_r;
		IF n < HLI_KEY_MAXIDX THEN
			n := n+1;
		END_IF
	END_IF
END_FOR

END_FUNCTION

// ---- CNC Beckhoff/2 OperationMode/ModeManual/PRG_AnalogJoystick.TcPOU
PROGRAM PRG_AnalogJoystick
VAR_INPUT
	nLogAxisNr: UINT;
	/// Actual Analog Value 
	Analog_Value: DINT;
	/// static signal : Analog Min Value 
	AnalogValueMin: DINT;
	/// static signal : Analog Max Value 
	AnalogValueMax: DINT;
	/// Dead Band for Zero Value 
	AnalogValueZeroDeadBand: DINT;
END_VAR
VAR_IN_OUT
	bKeyPos: BOOL;
	bKeyNeg: BOOL;
END_VAR
VAR
	/// Index of axis specific HLI area 
	nHliAxisIdx: INT;
	Norm_AnalogValue: LREAL;
	Zero_AnalogValue: LREAL;
	Override: LREAL;
END_VAR

(* ========================================================= *)
(*    Prog: Analog JoyStick			                  		 *)
(* --------------------------------------------------------- *)
(*   Desc:                                                   *)
(*   Author: TV	, MiB	                                         *)
(*   Date: 24.07.2015                                       *)
(*   Rev.: 6.0                                               *)
(* ========================================================= *)
	Norm_AnalogValue := (AnalogValueMax - AnalogValueMin);
	Zero_AnalogValue := AnalogValueMin + Norm_AnalogValue / 2;

	IF nLogAxisNr > 0 AND Norm_AnalogValue > 0 THEN
		nHliAxisIdx :=  HLI3_GetHliAxisIdx(UINT_TO_INT(nLogAxisNr));
		IF (nHliAxisIdx = -1) THEN
			RETURN;
		END_IF
		gpAx[nHliAxisIdx]^.ipo_mc_control.override.enable_w := TRUE;
		gpAx[nHliAxisIdx]^.ipo_mc_control.override_valid.enable_w := TRUE;
		gpAx[nHliAxisIdx]^.ipo_mc_control.override_valid.command_w := TRUE;
		Override := ABS(((Analog_Value  - AnalogValueMin) * 200 / Norm_AnalogValue)-100);

		IF Override > 100.0 THEN Override := 100.0; END_IF

		IF Analog_Value > Zero_AnalogValue THEN bKeyPos := TRUE; bKeyNeg := FALSE; ELSE bKeyPos := FALSE; END_IF
		IF Analog_Value < Zero_AnalogValue THEN bKeyNeg := TRUE; bKeyPos := FALSE; ELSE bKeyNeg := FALSE; END_IF

		IF Analog_Value > (Zero_AnalogValue - AnalogValueZeroDeadBand) AND Analog_Value < (Zero_AnalogValue + AnalogValueZeroDeadBand) THEN
			Override := 0;
			bKeyNeg := FALSE;
			bKeyPos := FALSE;
		END_IF

		gpAx[nHliAxisIdx]^.ipo_mc_control.override.command_w := LREAL_TO_UINT(Override * 10);
	END_IF

END_PROGRAM

// ---- CNC Beckhoff/9 Mis/HLI3_GetHliAxisIdx.TcPOU
FUNCTION HLI3_GetHliAxisIdx : INT
VAR_INPUT
	nLogAxisId: INT;
END_VAR
VAR
	i: INT;
END_VAR

(* ========================================================= *)
(*    FUN: HLI3_GetHliAxisIdx                            *)
(* --------------------------------------------------------- *)
(*   Desc: returns teh HliAxisIdx for a given logical Axis id      	*)
(*   Author: MiB                                             *)
(*   Date: 19.11.2012                                        *)
(*   Rev.: 1.0                                               *)
(* ========================================================= *)
HLI3_GetHliAxisIdx := -1;
FOR i := 0 TO UDINT_TO_INT(gNrAx) DO
	IF nLogAxisId = UINT_TO_INT(gpAx[i]^.head.log_ax_nr_r) THEN
		HLI3_GetHliAxisIdx := i;
		RETURN;
	END_IF
END_FOR

END_FUNCTION

// ---- CNC Beckhoff/Messages/FB_ChannelError.TcPOU
FUNCTION_BLOCK FB_ChannelError
VAR_INPUT
	nChanIdx: INT;
END_VAR
VAR_OUTPUT
	Valid: BOOL := FALSE;
	/// Identification of channel error 
	ChErrorID: UDINT;
	/// Module name 
	ModuleName: STRING;
	/// Line in source file 
	Line: DINT;
	/// Multiple ID 
	MultipleID: DINT;
	/// Commandable function type 
	CmdFunctionType: DINT;
	/// Identification of the channel 
	ChannelID: DINT;
	/// Communication ID 
	CommuID: DINT;
	/// Cycle counter of CNC 
	CycleCounter: UDINT;
	/// Version name 
	VersionName: STRING;
	/// Remedy class of error 
	RemedyClass: DINT;
	/// Reaction class of error 
	ReactionClass: DINT;
	/// Body type of error 
	BodyType: UDINT;
	/// User message 
	UserMessage: STRING;
	/// Variables of error record body 
	BodyTypeEnum: UDINT;
	NcBlockNr: DINT := 0;
	ProgName: STRING := '';
	FileName: STRING := '';
	FileOffset: UDINT := 0;
	NcBlockOffset: DINT := 0;
	TokenOffset: DINT := 0;
	LogicalPathNr: DINT := 0;
	AddProgInfo: STRING := '';
	CommuMedium: DINT := 0;
	CommuType: UDINT := 0;
	CommuPartner: UDINT := 0;
	FileLine: UDINT := 0;
	ListType: DINT := 0;
	StructName: STRING := '';
	StrValue_1: STRING;
	StrValue_2: STRING;
	StrValue_3: STRING;
	StrValue_4: STRING;
	StrValue_5: STRING;
	MeaningValue_1: STRING;
	MeaningValue_2: STRING;
	MeaningValue_3: STRING;
	MeaningValue_4: STRING;
END_VAR
VAR
	/// Index of channel specific HLI area 	
	pMcError: POINTER TO MC_ERROR;
	
	pMcError2: POINTER TO MC_ERROR;
	SatzR: HLI_ERROR_SATZ;
	bInitialized: BOOL := FALSE;
	bClear: BOOL := FALSE;
	bUsed: ARRAY[0..CNC_EVENTS_MAXIDX] OF BOOL;
	bToCleanUp: ARRAY[0..CNC_EVENTS_MAXIDX] OF BOOL;
	LogEvent: ARRAY[0..CNC_EVENTS_MAXIDX] OF ADSLOGEVENT;
	FlankeQuit: ARRAY[0..CNC_EVENTS_MAXIDX] OF R_TRIG;
	pLog: POINTER TO ADSLOGEVENT;
	fmtStr: STRING;
	eventId: UDINT;
	i: UDINT;
	idx: UDINT := 0;
	maxWarnings: UINT;
	maxErrors: UINT;
	maxUserEvents: UINT;
	/// Gesamtzahl = Userevents und Errors 
	maxEvents: UINT;
	/// maximal index of an event 
	maxIdxEvents: UINT;
	countWarnings: UINT := 0;
	countErrors: UINT := 0;
	countUserEvents: UINT := 0;
	start_idx: UINT;
	stop_idx: UINT;
	paraPointerArray: ARRAY[0..31] OF POINTER TO UDINT;
	paraIndex: INT;
	pRumpfNcProg: POINTER TO HLI_RUMPF_NC_PROG;
	pRumpfNcProgLr: POINTER TO HLI_RUMPF_NC_PROG_LR;
	pRumpfMds: POINTER TO HLI_RUMPF_MDS;
	pRumpfKommu: POINTER TO HLI_RUMPF_KOMMU;
	pRumpfRamDisk: POINTER TO HLI_RUMPF_RAMDISK;
	pRumpfFile: POINTER TO HLI_RUMPF_FILE;
	pRumpfIntprFile: POINTER TO HLI_RUMPF_INTPR_FILE;
	pRumpfListeBinaer: POINTER TO HLI_RUMPF_LISTE_BINAER;
	pRumpfGcm: POINTER TO HLI_RUMPF_GCM;
	bTcComError: BOOL;	
	bAxisErr : BOOL; 
END_VAR
VAR CONSTANT
	XmlEventId_Rumpf: UDINT := 200;
	XmlEventId_RumpfNcProg: UDINT := 201;
	XmlEventId_RumpfNcProgLr: UDINT := 202;
	XmlEventId_RumpfMds: UDINT := 203;
	XmlEventId_RumpfKommu: UDINT := 204;
	XmlEventId_RumpfRamDisk: UDINT := 205;
	XmlEventId_RumpfFile: UDINT := 206;
	XmlEventId_RumpfIntprFile: UDINT := 207;
	XmlEventId_RumpfListeBinaer: UDINT := 208;
	XmlEventId_RumpfGcm: UDINT := 209;
	CNC_SOURCE_ID_BASE: UDINT := 551;
	CNC_USER_SOURCE_ID_BASE: UDINT := 651;
	MAX_CNC_ERRORS: UDINT := 49;
	MAX_CNC_USER_EVENTS: UDINT := 49;
	/// MAX_CNC_ERRORS + MAX_CNC_USER_EVENTS 
	MAX_CNC_EVENTS: UDINT := 98;
	/// MAX_CNC_EVENTS - 1 
	CNC_EVENTS_MAXIDX: UDINT := 97;
	ERR_BAHN_ONLINE_TRC_CALCULATION: UDINT := 50689;
	ERR_ID_REPORT_CNC_RESET: UDINT := 270076;
	ERR_ID_KIN_TRAFO_CONFIG: UDINT := 292030;
	ERR_ID_KIN_TRAFO_INIT: UDINT := 292031;
	ERR_ID_KIN_TRAFO_FORWARD: UDINT := 292032;
	ERR_ID_KIN_TRAFO_BACKWARD: UDINT := 292033;
END_VAR

(* ========================================================= *)
(*    FB: FB_ChannelError                               	 *)
(* --------------------------------------------------------- *)
(*   Desc: FB transfers CNC Errors to the Event Logger		 *)
(*   Author: ISG / TV                                        *)
(*   Date: 12.10.2015                                        *)
(*   Rev.: 1.3                                              *)
(*															 *)
(* ========================================================= *)

(* check for channel no *)
IF NOT HLI3_CheckChannelValid(nChannel := nChanIdx) THEN
	RETURN;
END_IF

(* check for zero pointer *)
IF gpCh[nChanIdx] = 0 THEN
  RETURN;
END_IF

(* check for zero pointer, first channel is necessary for axis errors (Position controller errors) *)
IF gpCh[0] = 0 THEN
  RETURN;
END_IF

pMcError := ADR(gpCh[nChanIdx]^.mc_error);
SatzR    := pMcError^.satz_r;

IF bInitialized = FALSE THEN
  pMcError^.enable_w := TRUE;    (* enable control unit for error messages *) 
  bInitialized  := TRUE;
  maxErrors     := UDINT_TO_UINT(MAX_CNC_ERRORS / gNrCh);
  maxWarnings   := maxErrors / 5;
  maxUserEvents := UDINT_TO_UINT(MAX_CNC_USER_EVENTS / gNrCh);
  maxEvents     := maxUserEvents + maxErrors;

  maxIdxEvents := (maxEvents - 1);
  FOR i := 0 TO maxIdxEvents DO
    (* ----------------------------------------- *)
    (* initialize fixed elements of event        *)
    (* ----------------------------------------- *)
    pLog := ADR( LogEvent[i] );
    pLog^.NETID := '';      (* Local Computer *)
    pLog^.PORT:= 110;       (* Event Logger *)
    pLog^.TMOUT:= t#10s;
    pLog^.EventConfigData.Prio         := TCEVENTPRIO_IMPLICIT;
    pLog^.EventConfigData.ProgId       := 'TcEventFormatter.TcXmlFormatter';
    pLog^.EventConfigData.Flags        := TCEVENTFLAG_SRCID OR TCEVENTFLAG_LOG;
    pLog^.EventConfigData.SourceString := '';
    pLog^.EventConfigData.StreamType   := TCEVENTSTREAM_NORMAL;

    IF i < maxErrors THEN
      (* SourceID: 550 error texts, [ 551,  599] for single CNC error messages *)
      pLog^.EventConfigData.SourceId := CNC_SOURCE_ID_BASE + i + (DINT_TO_UINT(nChanIdx)*maxErrors);
    ELSE
      (* SourceID: 650 user error texts, [ 651,  699] for single CNC user error messages "ERROR[]" *)
      pLog^.EventConfigData.SourceId := CNC_USER_SOURCE_ID_BASE + i-maxErrors + (DINT_TO_UINT(nChanIdx)*maxUserEvents);
    END_IF

    FlankeQuit[i](CLK :=  pLog^.Quit);
  END_FOR
END_IF



(* -------------------------------------------------------------------------*)
(* test if events which have been reported shall be cleared again           *)
(* -------------------------------------------------------------------------*)
IF bClear THEN
  bClear := FALSE;
  countWarnings := 0;
  countErrors := 0;
  countUserEvents := 0;
  FOR i := 0 TO maxIdxEvents DO
    IF bToCleanup[i] = FALSE AND bUsed[i] THEN
      bToCleanup[i] := TRUE;
    END_IF
  END_FOR
END_IF


(* -------------------------------------------------------------------------*)
(* check for new error message                                              *)
(* -------------------------------------------------------------------------*)

(* Output for position controller errors is gpCh[0]^ *)
IF gpCh[0]^.mc_error.semaphor_rw THEN	
	SatzR := gpCh[0]^.mc_error.satz_r;		
	bAxisErr := TRUE;				
END_IF

IF (pMcError^.semaphor_rw  OR bAxisErr)  THEN

 	IF  SatzR.kopf.cnc_channel > 0 THEN 
  		IF (SatzR.kopf.cnc_channel-1 <> INT_TO_UINT(nChanIdx)) THEN	  
			bAxisErr := FALSE;		
    	RETURN;
	END_IF
  END_IF
  
  (* Initialize output variables that depend on error body type *)
  NcBlockNr      := 0;
  ProgName       := '';
  FileName       := '';
  FileOffset     := 0;
  NcBlockOffset  := 0;
  TokenOffset    := 0;
  LogicalPathNr  := 0;
  AddProgInfo    := '';

  CommuMedium    := 0;
  CommuType      := 0;
  CommuPartner   := 0;

  FileLine       := 0;
  ListType       := 0;
  StructName     := '';

  StrValue_1     := '';
  StrValue_2     := '';
  StrValue_3     := '';
  StrValue_4     := '';
  StrValue_5     := '';

  MeaningValue_1 := '';
  MeaningValue_2 := '';
  MeaningValue_3 := '';
  MeaningValue_4 := '';


  eventId := SatzR.kopf.error_id;

  (*------------------------------------------------------------------*)
  (* automatic clear old events if CNC reports reset                  *)
  (*------------------------------------------------------------------*)
  IF eventId = ERR_ID_REPORT_CNC_RESET THEN
	  	IF bAxisErr THEN 
    		gpCh[0]^.mc_error.semaphor_rw := FALSE;
			bAxisErr := FALSE;
		ELSE
			pMcError^.semaphor_rw := FALSE;		
		END_IF
	
    bClear := TRUE;
    RETURN;
  END_IF

  
  (*------------------------------------------------------------------*)
  (* TcCom: kinematic transformation, map util_error_id to error_id   *)
  (*------------------------------------------------------------------*)
  IF    eventId = ERR_ID_KIN_TRAFO_CONFIG
     OR eventId = ERR_ID_KIN_TRAFO_INIT  
     OR eventId = ERR_ID_KIN_TRAFO_FORWARD
     OR eventId = ERR_ID_KIN_TRAFO_BACKWARD
   OR eventId = ERR_BAHN_ONLINE_TRC_CALCULATION
  THEN
    eventId := SatzR.kopf.util_error_id;
    bTcComError := TRUE;
  ELSE
    bTcComError := FALSE;
  END_IF
   

  (*-------------------------------*)
  (* search unused event           *)
  (*-------------------------------*)
  IF eventId <= 1000 OR bTcComError THEN
    countUserEvents := countUserEvents + 1;
    start_idx       := maxErrors;
    stop_idx        := maxErrors + maxUserEvents - 1;
  ELSE
    (*------------------------------------------------------------------*)
    (* check maximum number of active warnings                          *)
    (*------------------------------------------------------------------*)
    IF SatzR.kopf.behebungs_klasse < 2 THEN
      IF countWarnings > maxWarnings THEN
		  IF (bAxisErr) THEN
			  	gpCh[0]^.mc_error.semaphor_rw := FALSE;
				bAxisErr := FALSE;
		  ELSE	
				pMcError^.semaphor_rw := FALSE;	  
		  END_IF
        
        RETURN;  (* dismiss further warning *)
      END_IF
      countWarnings:= countWarnings + 1;
    END_IF

    countErrors := countErrors + 1;
    start_idx   := 0;
    stop_idx    := maxErrors - 1;
  END_IF

  FOR i := start_idx TO stop_idx DO
    IF bUsed[i] = FALSE THEN
      EXIT;
    END_IF
  END_FOR

  IF i > stop_idx THEN
    (*------------------------------------------------------------------*)
    (* overflow -> dismiss actual message, wait for reset               *)
    (*------------------------------------------------------------------*)
	IF (bAxisErr) THEN
		gpCh[0]^.mc_error.semaphor_rw := FALSE;
		bAxisErr := FALSE;
	ELSE	
		pMcError^.semaphor_rw := FALSE;	  
	END_IF	
    RETURN;
  END_IF
  idx := i;


  bUsed[idx] := TRUE;
  pLog := ADR( LogEvent[idx] );

  (* Initialisierungen fuer jeden Aufruf *)
  paraIndex := 0;

  (*
    TCEVENTCLASS_NONE        := 0,  No class
    TCEVENTCLASS_MAINTENANCE := 1,  Maintenance hint
    TCEVENTCLASS_MESSAGE     := 2,  Message
    TCEVENTCLASS_HINT        := 3,  Hint
    TCEVENTCLASS_STATEINFO   := 4,  State information
    TCEVENTCLASS_INSTRUCTION := 5,  Instruction
    TCEVENTCLASS_WARNING     := 6,  Warning
    TCEVENTCLASS_ALARM       := 7,  Alarm
    TCEVENTCLASS_PARAMERROR
  *)

  IF SatzR.kopf.behebungs_klasse < 2 THEN
    pLog^.EventConfigData.Class := TCEVENTCLASS_WARNING;
    pLog^.EventConfigData.bQuitRequired := FALSE;  (* Hasn't to acknowledge the event *)
  ELSE
    pLog^.EventConfigData.bQuitRequired := TRUE;  (* Has to acknowledge the event *)
    IF SatzR.kopf.behebungs_klasse < 7 THEN
      pLog^.EventConfigData.Class := TCEVENTCLASS_ALARM;
    ELSE
      pLog^.EventConfigData.Class := TCEVENTCLASS_PARAMERROR;
    END_IF
  END_IF
  pLog^.EventConfigData.Id := XmlEventId_Rumpf;

  (*------------------------------------------------------------------*)
  (* parameters 1 - 13 are content independent                        *)
  (*------------------------------------------------------------------*)
  fmtStr := '%d%d%d%d%s%d%d%d%d%d%s%d%s';  (* a string *)

  (* If ChErrorID has a link to a sub string (other EventId and SourceId)  *)
  (* a string is build of following syntax: '[SxEy]' with x as SourceId and y as EventId *)
  (* in TcCncError.xml x alsways has value 2 and y is the ChErrorID of the CNC *)
  (* ----------------------------------------------------*)
  (* User specific error message                         *)
  (* ----------------------------------------------------*)
  IF eventId <= 1000 OR bTcComError THEN
    UserMessage   := '[S650E'; (* sub string from SourceId 550 (see TcCncUserEvents.xml) and EventId 'eventId' *)
  ELSE
    UserMessage   := '[S550E'; (* sub string from SourceId 2 (see TcCncError.xml) and EventId 'eventId' *)
  END_IF
  UserMessage     := CONCAT(UserMessage, UDINT_TO_STRING(eventId));
  UserMessage     := CONCAT(UserMessage, ']');

  ChErrorID       := eventId;
  ChannelID       := SatzR.kopf.cnc_channel;
  RemedyClass     := SatzR.kopf.behebungs_klasse;
  ReactionClass   := SatzR.kopf.reaktions_klasse;
  ModuleName      := SatzR.kopf.modul_name.zeichen;
  Line            := SatzR.kopf.line;
  MultipleID      := SatzR.kopf.multiple_id;
  CmdFunctionType := SatzR.kopf.bf_type;

  CommuID         := SatzR.kopf.kommu_id;
  CycleCounter    := SatzR.kopf.fb_zeitangabe.zykl_counter;
  VersionName     := SatzR.kopf.version_name.zeichen;
  BodyType        := SatzR.kopf.rumpf_typ;

  paraPointerArray[paraIndex] := ADR(ChErrorID);
  paraIndex := paraIndex + 1;
  paraPointerArray[paraIndex] := ADR(ChannelID);
  paraIndex := paraIndex + 1;
  paraPointerArray[paraIndex] := ADR(RemedyClass);
  paraIndex := paraIndex + 1;
  paraPointerArray[paraIndex] := ADR(ReactionClass);
  paraIndex := paraIndex + 1;
  paraPointerArray[paraIndex] := ADR(ModuleName);
  paraIndex := paraIndex + 1;
  paraPointerArray[paraIndex] := ADR(Line);
  paraIndex := paraIndex + 1;
  paraPointerArray[paraIndex] := ADR(MultipleID);
  paraIndex := paraIndex + 1;
  paraPointerArray[paraIndex] := ADR(CmdFunctionType);
  paraIndex := paraIndex + 1;
  paraPointerArray[paraIndex] := ADR(CommuID);
  paraIndex := paraIndex + 1;
  paraPointerArray[paraIndex] := ADR(CycleCounter);
  paraIndex := paraIndex + 1;
  paraPointerArray[paraIndex] := ADR(VersionName);
  paraIndex := paraIndex + 1;
  paraPointerArray[paraIndex] := ADR(BodyType);
  paraIndex := paraIndex + 1;
  paraPointerArray[paraIndex] := ADR(UserMessage);
  paraIndex := paraIndex + 1;


  (*------------------------------------------------------------------------*)
  (* Append values and meaning of values.                                   *)
  (*------------------------------------------------------------------------*)
  StrValue_1 := WertBToString(SatzR.rumpf.wert_1, 1);
  StrValue_2 := WertBToString(SatzR.rumpf.wert_2, 2);
  StrValue_3 := WertBToString(SatzR.rumpf.wert_3, 3);
  StrValue_4 := WertBToString(SatzR.rumpf.wert_4, 4);
  StrValue_5 := WertBToString(SatzR.rumpf.wert_5, 5);

  paraPointerArray[paraIndex] := ADR(StrValue_1);
  paraIndex := paraIndex + 1;
  paraPointerArray[paraIndex] := ADR(StrValue_2);
  paraIndex := paraIndex + 1;
  paraPointerArray[paraIndex] := ADR(StrValue_3);
  paraIndex := paraIndex + 1;
  paraPointerArray[paraIndex] := ADR(StrValue_4);
  paraIndex := paraIndex + 1;
  paraPointerArray[paraIndex] := ADR(StrValue_5);
  paraIndex := paraIndex + 1;

  fmtStr := CONCAT(fmtStr, '%s%s%s%s%s');

  MeaningValue_1 := WertToString(SatzR.rumpf.kennung_1, 1);
  MeaningValue_2 := WertToString(SatzR.rumpf.kennung_2, 2);
  MeaningValue_3 := WertToString(SatzR.rumpf.kennung_3, 3);
  MeaningValue_4 := WertToString(SatzR.rumpf.kennung_4, 4);

  paraPointerArray[paraIndex] := ADR(MeaningValue_1);
  paraIndex := paraIndex + 1;
  paraPointerArray[paraIndex] := ADR(MeaningValue_2);
  paraIndex := paraIndex + 1;
  paraPointerArray[paraIndex] := ADR(MeaningValue_3);
  paraIndex := paraIndex + 1;
  paraPointerArray[paraIndex] := ADR(MeaningValue_4);
  paraIndex := paraIndex + 1;

  fmtStr := CONCAT(fmtStr, '%s%s%s%s');



  BodyTypeEnum := SatzR.kopf.rumpf_typ;

  (*-------------------------------------------------------------------------*)
  (*       HLI_RUMPF_TYP_NC_PROG                                             *)
  (*-------------------------------------------------------------------------*)
  IF BodyTypeEnum = HLI_RUMPF_TYP_NC_PROG THEN
    pLog^.EventConfigData.Id := XmlEventId_RumpfNcProg;

    pRumpfNcProg := ADR(SatzR.rumpf.maske);

    (* Assign error body data to output variables *)
    NcBlockNr     := pRumpfNcProg^.satz_nr;
    ProgName      := pRumpfNcProg^.prog_name.zeichen;
    FileName      := pRumpfNcProg^.file_name.zeichen;
    FileOffset    := pRumpfNcProg^.fileoffset;
    NcBlockOffset := pRumpfNcProg^.satzoffset;
    TokenOffset   := pRumpfNcProg^.tokenoffset;
    LogicalPathNr := pRumpfNcProg^.log_pfad_nr;
    AddProgInfo   := pRumpfNcProg^.add_prog_info.zeichen;

    (* Assign address of data to parameter array of the event *)
    paraPointerArray[paraIndex] := ADR(NcBlockNr);
    paraIndex := paraIndex + 1;
    paraPointerArray[paraIndex] := ADR(ProgName);
    paraIndex := paraIndex + 1;
    paraPointerArray[paraIndex] := ADR(FileName);
    paraIndex := paraIndex + 1;
    paraPointerArray[paraIndex] := ADR(FileOffset);
    paraIndex := paraIndex + 1;
    paraPointerArray[paraIndex] := ADR(NcBlockOffset);
    paraIndex := paraIndex + 1;
    paraPointerArray[paraIndex] := ADR(TokenOffset);
    paraIndex := paraIndex + 1;
    paraPointerArray[paraIndex] := ADR(LogicalPathNr);
    paraIndex := paraIndex + 1;
    paraPointerArray[paraIndex] := ADR(AddProgInfo);
    paraIndex := paraIndex + 1;

    (* Add format string for error messages out of NC programs *)
    fmtStr := CONCAT(fmtStr, '%d%s%s%d%d%d%d%s');
  (*-------------------------------------------------------------------------*)
  (*       HLI_RUMPF_TYP_NC_PROG_LR                                          *)
  (*-------------------------------------------------------------------------*)
  ELSIF BodyTypeEnum = HLI_RUMPF_TYP_NC_PROG_LR THEN
    pLog^.EventConfigData.Id := XmlEventId_RumpfNcProgLR;

    pRumpfNcProgLr := ADR(SatzR.rumpf.maske);

    LogicalPathNr  := pRumpfNcProgLr^.log_pfad_nr;
    ProgName       := pRumpfNcProgLr^.prog_name.zeichen;
    FileName       := pRumpfNcProgLr^.file_name.zeichen;
    NcBlockNr      := pRumpfNcProgLr^.satz_nr;
    AddProgInfo    := pRumpfNcProgLr^.add_prog_info.zeichen;

    paraPointerArray[paraIndex] := ADR(NcBlockNr);
    paraIndex := paraIndex + 1;
    paraPointerArray[paraIndex] := ADR(ProgName);
    paraIndex := paraIndex + 1;
    paraPointerArray[paraIndex] := ADR(FileName);
    paraIndex := paraIndex + 1;
    paraPointerArray[paraIndex] := ADR(LogicalPathNr);
    paraIndex := paraIndex + 1;
    paraPointerArray[paraIndex] := ADR(AddProgInfo);
    paraIndex := paraIndex + 1;

    fmtStr := CONCAT(fmtStr, '%d%s%s%d%s');
  (*-------------------------------------------------------------------------*)
  (*       HLI_RUMPF_TYP_MDS                                                 *)
  (*-------------------------------------------------------------------------*)
  ELSIF BodyTypeEnum = HLI_RUMPF_TYP_MDS THEN
    pLog^.EventConfigData.Id := XmlEventId_RumpfMds;

    pRumpfMds     := ADR(SatzR.rumpf.maske);

    LogicalPathNr := pRumpfMds^.listen_typ;
    ProgName      := pRumpfMds^.strukt_name.zeichen;

    paraPointerArray[paraIndex] := ADR(LogicalPathNr);
    paraIndex := paraIndex + 1;
    paraPointerArray[paraIndex] := ADR(ProgName);
    paraIndex := paraIndex + 1;

    fmtStr := CONCAT(fmtStr, '%d%s');
  (*-------------------------------------------------------------------------*)
  (*       HLI_RUMPF_TYP_KOMMU                                               *)
  (*-------------------------------------------------------------------------*)
  ELSIF BodyTypeEnum = HLI_RUMPF_TYP_KOMMU THEN
    pLog^.EventConfigData.Id := XmlEventId_RumpfKommu;

    pRumpfKommu  := ADR(SatzR.rumpf.maske);

    CommuMedium  := pRumpfKommu^.Medium;
    CommuType    := pRumpfKommu^.Typ;
    CommuPartner := pRumpfKommu^.Partner;

    paraPointerArray[paraIndex] := ADR(CommuMedium);
    paraIndex := paraIndex + 1;
    paraPointerArray[paraIndex] := ADR(CommuType);
    paraIndex := paraIndex + 1;
    paraPointerArray[paraIndex] := ADR(CommuPartner);
    paraIndex := paraIndex + 1;

    fmtStr := CONCAT(fmtStr, '%d%d%d');
  (*-------------------------------------------------------------------------*)
  (*       HLI_RUMPF_TYP_RAMDISK                                             *)
  (*-------------------------------------------------------------------------*)
  ELSIF BodyTypeEnum = HLI_RUMPF_TYP_RAMDISK THEN
    pLog^.EventConfigData.Id := XmlEventId_RumpfRamDisk;

    pRumpfRamDisk := ADR(SatzR.rumpf.maske);

    CommuMedium   := pRumpfRamDisk^.medium;
    CommuType     := pRumpfRamDisk^.typ;
    CommuPartner  := pRumpfRamDisk^.partner;
    FileName      := pRumpfRamDisk^.file_name.zeichen;
    FileOffset    := pRumpfRamDisk^.fileoffset;

    paraPointerArray[paraIndex] := ADR(CommuMedium);
    paraIndex := paraIndex + 1;
    paraPointerArray[paraIndex] := ADR(CommuType);
    paraIndex := paraIndex + 1;
    paraPointerArray[paraIndex] := ADR(CommuPartner);
    paraIndex := paraIndex + 1;
    paraPointerArray[paraIndex] := ADR(FileName);
    paraIndex := paraIndex + 1;
    paraPointerArray[paraIndex] := ADR(FileOffset);
    paraIndex := paraIndex + 1;

    fmtStr := CONCAT(fmtStr, '%d%d%d%s%d');
  (*-------------------------------------------------------------------------*)
  (*       HLI_RUMPF_TYP_FILE                                                *)
  (*-------------------------------------------------------------------------*)
  ELSIF BodyTypeEnum = HLI_RUMPF_TYP_FILE THEN
    pLog^.EventConfigData.Id := XmlEventId_RumpfFile;

    pRumpfFile := ADR(SatzR.rumpf.maske);

    FileName   := pRumpfFile^.file_name.zeichen;
    FileOffset := pRumpfFile^.fileoffset;

    paraPointerArray[paraIndex] := ADR(FileName);
    paraIndex := paraIndex + 1;
    paraPointerArray[paraIndex] := ADR(FileOffset);
    paraIndex := paraIndex + 1;

    fmtStr := CONCAT(fmtStr, '%s%d');
  (*-------------------------------------------------------------------------*)
  (*       HLI_RUMPF_TYP_INTPR_FILE                                          *)
  (*-------------------------------------------------------------------------*)
  ELSIF BodyTypeEnum = HLI_RUMPF_TYP_INTPR_FILE THEN
    pLog^.EventConfigData.Id := XmlEventId_RumpfIntprFile;

    pRumpfIntprFile := ADR(SatzR.rumpf.maske);

    FileName   := pRumpfIntprFile^.file_name.zeichen;
    FileOffset := pRumpfIntprFile^.fileoffset;
    FileLine   := pRumpfIntprFile^.file_line_number;
    ListType   := pRumpfIntprFile^.listen_typ;
    StructName := pRumpfIntprFile^.strukt_name.zeichen;

    paraPointerArray[paraIndex] := ADR(FileName);
    paraIndex := paraIndex + 1;
    paraPointerArray[paraIndex] := ADR(FileOffset);
    paraIndex := paraIndex + 1;
    paraPointerArray[paraIndex] := ADR(FileLine);
    paraIndex := paraIndex + 1;
    paraPointerArray[paraIndex] := ADR(ListType);
    paraIndex := paraIndex + 1;
    paraPointerArray[paraIndex] := ADR(StructName);
    paraIndex := paraIndex + 1;

    fmtStr := CONCAT(fmtStr, '%s%d%d%d%s');
  (*-------------------------------------------------------------------------*)
  (*       HLI_RUMPF_TYP_LISTE_BINAER                                        *)
  (*-------------------------------------------------------------------------*)
  ELSIF BodyTypeEnum = HLI_RUMPF_TYP_LISTE_BINAER THEN
    pLog^.EventConfigData.Id := XmlEventId_RumpfListeBinaer;

    pRumpfListeBinaer := ADR(SatzR.rumpf.maske);

    StructName:=pRumpfListeBinaer^.strukt_name.zeichen;

    paraPointerArray[paraIndex] := ADR(StructName);
    paraIndex := paraIndex + 1;

    fmtStr := CONCAT(fmtStr, '%s');
  (*-------------------------------------------------------------------------*)
  (*       HLI_RUMPF_TYP_GCM                                                 *)
  (*-------------------------------------------------------------------------*)
  ELSIF BodyTypeEnum = HLI_RUMPF_TYP_GCM THEN
    pLog^.EventConfigData.Id := XmlEventId_RumpfGcm;

    pRumpfGcm := ADR(SatzR.Rumpf.Maske);

    ProgName:=pRumpfGcm^.Token.zeichen;
    FileName:=pRumpfGcm^.FileName.zeichen;

    paraPointerArray[paraIndex] := ADR(ProgName);
    paraIndex := paraIndex + 1;
    paraPointerArray[paraIndex] := ADR(FileName);
    paraIndex := paraIndex + 1;

    fmtStr := CONCAT(fmtStr, '%s%s');
  END_IF

  (*------------------------------------------------------------------------*)
  (* Set values at input pins of FB                                         *)
  (*------------------------------------------------------------------------*)
  pLog^.EventDataAddress:= ADR(paraPointerArray);
  pLog^.EventDataLength:= 0;
  pLog^.fbCleanUp  := FALSE;
  pLog^.EventQuit  := FALSE;

  pLog^.EventConfigData.DataFormatStrAddress := ADR(fmtStr);

  (*------------------------------------------------------------------------*)
  (* report error message to event logger                                   *)
  (*------------------------------------------------------------------------*)
  pLog^(Event := TRUE);

  (* Notify at output that a error essage occurred *)
  Valid := TRUE;

  (* Acknowledge error message *)
 	IF (bAxisErr) THEN
		gpCh[0]^.mc_error.semaphor_rw := FALSE;
		bAxisErr := FALSE;
	ELSE	
		pMcError^.semaphor_rw := FALSE;	  
	END_IF
ELSE
  Valid := FALSE;
END_IF

(* by default : no error message is present, first search for error messages *)
FOR i := 0 TO maxIdxEvents DO
  (*-------------------------------------------------------------------------*)
  (*       clear event                                                       *)
  (*-------------------------------------------------------------------------*)
  IF bToCleanup[i] THEN
    pLog := ADR( LogEvent[i] );
    pLog^();

    IF pLog^.EventState=TCEVENTSTATE_SIGNALED THEN
      pLog^( Event:=FALSE);
    ELSIF pLog^.EventState=TCEVENTSTATE_RESET THEN
      pLog^( EventQuit:= TRUE);
    ELSIF pLog^.EventState=TCEVENTSTATE_CONFIRMED OR pLog^.EventState=TCEVENTSTATE_INVALID THEN
      (*pLog^( FbCleanup:= TRUE); bugfix 12.7.2005*)
      bUsed[i]     := FALSE;
      bToCleanup[i] := FALSE;
    END_IF;
  (*-------------------------------------------------------------------------*)
  (*       report event                                                      *)
  (*-------------------------------------------------------------------------*)
  ELSIF bUsed[i] THEN
    pLog := ADR( LogEvent[i] );
    pLog^();

    (* IF pLog^.EventConfigData.bQuitRequired = FALSE THEN
      FlankeQuit[i](CLK :=  pLog^.Quit);
      IF FlankeQuit[i].Q = TRUE THEN
        bUsed[i] := FALSE;
        QuitCount := QuitCount + 1;
      END_IF
    END_IF*)
  END_IF
END_FOR

END_FUNCTION_BLOCK

// ---- CNC Beckhoff/3 Control/HLI3_SetChannelOverride.TcPOU
FUNCTION HLI3_SetChannelOverride : BOOL
VAR_INPUT
	/// Number of channel 
	nChanIdx: INT;
	nOverride: UINT;
END_VAR

(* ========================================================= *)
(*    FUN: HLI_SetChannelOverride                            *)
(* --------------------------------------------------------- *)
(*   Desc: Set the channel Override                          *)
(* Author: MK, MiB                                           *)
(*   Date: 20.11.2012                                        *)
(*   Rev.: 1.1                                               *)
(* ========================================================= *)

IF NOT HLI3_CheckChannelValid(nChannel := nChanIdx) THEN
	HLI3_SetChannelOverride := FALSE;
	RETURN;
END_IF

(* Limit the override *)
IF nOverride > 1200	THEN nOverride := 1200; END_IF
IF nOverride < 0 THEN nOverride := 0; END_IF

gpCh[nChanIdx]^.bahn_mc_control.override_feedrate.command_w := nOverride;

HLI3_SetChannelOverride := TRUE;

END_FUNCTION

// ---- CNC Beckhoff/PRG_CNCVariablesViewer.TcPOU
PROGRAM PRG_CNCVariablesViewer
VAR			
	fbReadCNCVariables : FB_ReadCNCVariables;		
END_VAR

fbReadCNCVariables(
	bEnable:= TRUE, 
	nChanIdx:= PLCSelectedChannel-1, 
	eVariablesType:= eVariablesType, 
	tIntervall:= T#1S, 	 
	stCNCVariablesViewer_Data:= stCNCVariablesViewer_Data);

END_PROGRAM

// ---- CNC Beckhoff/5 Variables/FB_ReadCNCVariables.TcPOU
FUNCTION_BLOCK FB_ReadCNCVariables
VAR_INPUT
	bEnable		:	BOOL ;	(* B *)
	nChanIdx	:   INT;
	eVariablesType : E_CNCVariablesType;
	tIntervall	:   TIME;
END_VAR

VAR_OUTPUT
	Done			:	BOOL;	(* B *)
	Busy			: 	BOOL;	(* E *)	
	Error			:	BOOL;	(* B *)
	ErrorID			:	UDINT;	(* E *) 
END_VAR

VAR_IN_OUT
	 stCNCVariablesViewer_Data : ARRAY[0..MAX_CNC_VAR_LIST_IDX] OF ST_CNCVariablesViewer_Data;
END_VAR

VAR	
	fbTrigger :	R_TRIG;
	fbReadNumber: ADSREAD;
	nParameterNumber : DINT;
		
	fbReadWrite: ADSRDWRT;	
	strVarName : STRING(96);	
	fVarValue  : LREAL;    
 	nIndex     : UDINT;
	nListIndex : UDINT;	
	
	nState	: INT;
	fbTimer : TON;

	nReadLength 	   : UDINT;
	
 	IDXOffsNumber	   : UDINT;
	IDXOffsNamebyIndex : UDINT;
	IDXOffsValuebyIndex : UDINT;	
	stCNCVariablesViewer_Data_Temp : ARRAY[0..MAX_CNC_VAR_LIST_IDX] OF ST_CNCVariablesViewer_Data;
		
	nVEType 				: DINT;
	nVESize 	 			: UDINT;
    nVEMaxIndex1 		   	: UDINT; 
    nVEMaxIndex2 		   	: UDINT;
	strVEVarName 			: STRING(255);	
	strVEDisplayVarName		: STRING(255);
	arrVEDescriptionInput  	: ARRAY[0..259] OF BYTE;
	arrVEOutput 			: ARRAY[0..2047] OF BYTE;
			
	nVEArrayIndex       	: UDINT;
	nListIndexArrayStart	: UDINT; 	
	
	strValue            : STRING(127);
			
	dummyBoolean		: BOOL;
	dummySInt			: SINT;
	dummyUSInt			: USINT;
	dummyInt            : INT;
	dummyUInt			: UINT;
	dummyDInt           : DINT;
	dummyUDInt          : UDINT;
	dummyLReal          : LREAL;
	dummyString         : STRING;
	dummyLargeString    : STRING(127);  

	eVariablesTypeOld : E_CNCVariablesType;
	
END_VAR

VAR CONSTANT
	IDXOffsPNumber  : UDINT := 16#2;	
	IDXOffsVLNumber : UDINT := 16#3;
	IDXOffsVPNumber : UDINT := 16#4;
	IDXOffsVSNumber : UDINT := 16#5;
			
	IDXOffsPNamebyIndex : UDINT := 16#1B;
	IDXOffsVLNamebyIndex : UDINT := 16#1E;
	IDXOffsVPNamebyIndex : UDINT := 16#21;
	IDXOffsVSNamebyIndex : UDINT := 16#24;		
	
	IDXOffsPValuebyIndex : UDINT := 16#1D;
	IDXOffsVLValuebyIndex : UDINT := 16#20;
	IDXOffsVPValuebyIndex : UDINT := 16#23;
	IDXOffsVSValuebyIndex : UDINT := 16#26;
	IDXOffsVEValuebyName : UDINT := 16#2E;		
END_VAR

(****************************************************************************************)
(* POU:		ReadCNCVariables                     										*)
(* Type:	FB																			*)
(* Author: 	TV                                             								*)
(* Date: 	20.01.2016																	*)
(* Rev.: 	1.0                                              							*)
(* ------------------------------------------------------------------------------------ *)
(* Desc:	Description																	*)
(****************************************************************************************)

(****************************************************************************************)
(*	FB reads in P, V.P, V.L., V.S., V.E. Parameter from the CNC Kernel via ADS		    *)
(****************************************************************************************)

IF (NOT HLI3_CheckChannelValid(nChannel := nChanIdx)) THEN	
	RETURN; (* A b b r u c h *)
END_IF

IF 	NOT bEnable OR 
	eVariablesType = E_CNCVariablesType.none  OR
	(gpCh[0]^.channel_mc_control.mode_and_state.state_r.mode = HLI_IMCM_MANUAL_MODE AND eVariablesType <> E_CNCVariablesType.VE) OR
	(gpCh[nChanIdx]^.channel_mc_control.mode_and_state.state_r.state <> HLI_IMCM_PROCESS_ACTIVE AND 
	gpCh[nChanIdx]^.channel_mc_control.mode_and_state.state_r.state <>  HLI_IMCM_PROCESS_HOLD AND eVariablesType <> E_CNCVariablesType.VE) 
		
	THEN
		Tc2_System.MEMSET(ADR(stCNCVariablesViewer_Data),0,SIZEOF(stCNCVariablesViewer_Data));
		fbTrigger(CLK:= FALSE);
		nState := 0;  
	ELSE
		fbTrigger(CLK:= TRUE);	
END_IF

IF fbTrigger.Q OR eVariablesTypeOld <> eVariablesType THEN		
	fbReadNumber(READ:= FALSE);
	fbReadWrite(WRTRD:= FALSE);
	nIndex 		:= 1;	
	nListIndex  := 0;
	nState 		:= 1;
	Error		:= FALSE;	(* B *)
	ErrorID		:= 0;		(* E *) 
END_IF

IF nState <> 0 THEN
	Busy := TRUE;
END_IF

CASE nState OF
	
0:
;  
1: 
	Error		:= FALSE;	(* B *)
	ErrorID		:= 0;	(* E *)

	eVariablesTypeOld :=  eVariablesType;
 
	Tc2_System.MEMSET(ADR(stCNCVariablesViewer_Data_Temp),0,SIZEOF(stCNCVariablesViewer_Data_Temp));
	
   	IF (eVariablesType = E_CNCVariablesType.P) THEN
	      IDXOffsNumber 	 	:= IDXOffsPNumber;
		  IDXOffsNamebyIndex 	:= IDXOffsPNamebyIndex;
		  IDXOffsValuebyIndex 	:= IDXOffsPValuebyIndex;
		  nReadLength			:= 8;			  
	ELSIF (eVariablesType = E_CNCVariablesType.VL) THEN
		 IDXOffsNumber 		 	:=  IDXOffsVLNumber;
		 IDXOffsNamebyIndex  	:= IDXOffsVLNameByIndex;
		 IDXOffsValuebyIndex 	:= IDXOffsVLValuebyIndex;
		 nReadLength			:= 8;
	ELSIF (eVariablesType = E_CNCVariablesType.VP) THEN
		 IDXOffsNumber 		 	:=  IDXOffsVPNumber;
		 IDXOffsNamebyIndex  	:= IDXOffsVPNameByIndex;
		 IDXOffsValuebyIndex 	:= IDXOffsVPValuebyIndex;
		 nReadLength			:= 8;
	ELSIF (eVariablesType = E_CNCVariablesType.VS) THEN
		 IDXOffsNumber 		 	:=  IDXOffsVSNumber;
		 IDXOffsNamebyIndex  	:= IDXOffsVSNameByIndex;
		 IDXOffsValuebyIndex 	:= IDXOffsVSValuebyIndex;
		 nReadLength			:= 8;	
   	END_IF
				
	
	IF (eVariablesType <> E_CNCVariablesType.VE) THEN
		fbReadNumber(
			NETID:= , 
			PORT:= 552, 
			IDXGRP:= 16#22300 + INT_TO_UDINT(nChanIdx)+1, 
			IDXOFFS:= IDXOffsNumber, 
			LEN:= 4, 
			DESTADDR:= ADR(nParameterNumber), 
			READ:= TRUE, 
		);
		
		IF NOT fbReadNumber.Busy THEN
			IF fbReadNumber.Err	THEN
				Error := fbReadNumber.ERR;
				ErrorID := fbReadNumber.ERRID;
				nState := 99;
			ELSE			
				nState := nState + 1;				
			END_IF
		END_IF
	ELSE
		nState := 20;
	END_IF

2:	// Read Variablen Name	
	IF nParameterNumber > 0 THEN 
		fbReadWrite(
		NETID:= , 
		PORT:= 552, 
		IDXGRP:= 16#22300 + INT_TO_UDINT(nChanIdx)+1, 
		IDXOFFS:= IDXOffsNamebyIndex, 
		WRITELEN:= 4, 
		READLEN:= 96, 
		SRCADDR:= ADR(nIndex), 
		DESTADDR:=ADR(strVarName), 
		WRTRD:= TRUE);
	
		IF NOT fbReadWrite.Busy THEN
			IF fbReadWrite.Err	THEN
				Error := fbReadWrite.ERR;
				ErrorID := fbReadWrite.ERRID;
				nState := 99;
			ELSE					
				fbReadWrite(WRTRD:= FALSE);	
				nState := 3;							
			END_IF
		END_IF
	
	ELSE	
		nState := 99;
	END_IF
	
	
3:	// Read Variablen Value	P V.L. V.P. V.S	
		fbReadWrite(
		NETID:= , 
		PORT:= 552, 
		IDXGRP:= 16#22300 + INT_TO_UDINT(nChanIdx)+1, 
		IDXOFFS:= IDXOffsValuebyIndex, 
		WRITELEN:= 4, 
		READLEN:= nReadLength, 
		SRCADDR:= ADR(nIndex), 
		DESTADDR:=ADR(fVarValue), 
		WRTRD:= TRUE);
	
		IF NOT fbReadWrite.Busy THEN
			IF fbReadWrite.Err	THEN
				Error := fbReadWrite.ERR;
				ErrorID := fbReadWrite.ERRID;
				nState := 99;
			ELSE
				stCNCVariablesViewer_Data_Temp[nListIndex].strName := strVarName;
				stCNCVariablesViewer_Data_Temp[nListIndex].strValue := LREAL_TO_STRING(fVarValue);		
				nListIndex := nListIndex+1;								
				nState := 4;
			END_IF
		END_IF		
		
		
4:  
	IF nIndex < DINT_TO_UDINT(nParameterNumber) AND (nListIndex <= MAX_CNC_VAR_LIST_IDX) THEN
		fbReadWrite(WRTRD:= FALSE);
		//nListIndex := nListIndex+1; 
		nIndex := nIndex + 1;
		nState := 2;
	ELSE
			fbTimer(IN:=FALSE);
			nState := 60;
	END_IF

20:    	// Read V.E. Variable element number
		arrVEDescriptionInput[0] := 86; // V
		arrVEDescriptionInput[1] := 46; //.
		arrVEDescriptionInput[2] := 69; //E
		
		fbReadWrite(
			NETID:= , 
			PORT:= 552, 
			IDXGRP:= 16#22300 + INT_TO_UDINT(nChanIdx)+1, 
			IDXOFFS:= 16#44, 
			WRITELEN:= 256, 
			READLEN:= 4, 
			SRCADDR:= ADR(arrVEDescriptionInput), 
			DESTADDR:=ADR(nParameterNumber), 
			WRTRD:= TRUE);

			IF NOT fbReadWrite.Busy THEN
				IF fbReadWrite.Err	THEN
					Error := fbReadWrite.ERR;
					ErrorID := fbReadWrite.ERRID;
					nState := 99;
				ELSE
					fbReadWrite(WRTRD:= FALSE);
					IF nParameterNumber > 0 THEN	
						nIndex := 0;		
						nListIndexArrayStart := 0;
						nVEArrayIndex := 0;			
						nState := 21;					
					ELSE			
						fbTimer(IN:=FALSE);
						nState := 60;			
					END_IF
				END_IF	
			END_IF			
			
21:		// Read V.E. Variable description by index
		MEMCPY(ADR(arrVEDescriptionInput),ADR(nIndex),SIZEOF(nIndex));
		arrVEDescriptionInput[4] := 86; // V
		arrVEDescriptionInput[5] := 46; //.
		arrVEDescriptionInput[6] := 69; //E
		
		fbReadWrite(
			NETID:= , 
			PORT:= 552, 
			IDXGRP:= 16#22300 + INT_TO_UDINT(nChanIdx)+1, 
			IDXOFFS:= 16#45, 
			WRITELEN:= 260, 
			READLEN:= 2048, 
			SRCADDR:= ADR(arrVEDescriptionInput), 
			DESTADDR:=ADR(arrVEOutput), 
			WRTRD:= TRUE);
	
		IF NOT fbReadWrite.Busy THEN
			IF fbReadWrite.Err	THEN
				Error := fbReadWrite.ERR;
				ErrorID := fbReadWrite.ERRID;
				nState := 99;
			ELSE
				fbReadWrite(WRTRD:= FALSE);
				
				//MEMCPY(ADR(nHandle),ADR(arrByte3),SIZEOF(nHandle));
				MEMCPY(ADR(nVEType),ADR(arrVEOutput)+4,SIZEOF(nVEType));
				// MEMCPY(ADR(nAccess),ADR(arrByte3)+4+4,SIZEOF(nAccess));
				MEMCPY(ADR(nVESize),ADR(arrVEOutput)+4+4+4,SIZEOF(nVESize));
				MEMCPY(ADR(nVEMaxIndex1),ADR(arrVEOutput)+4+4+4+4,SIZEOF(nVEMaxIndex1));
				IF nVEMaxIndex1 <> 0 THEN
					MEMCPY(ADR(nVEMaxIndex2),ADR(arrVEOutput)+4+4+4+4+4,SIZEOF(nVEMaxIndex2));
					MEMCPY(ADR(strVEVarName),ADR(arrVEOutput)+4+4+4+4+4+4,SIZEOF(strVEVarName));
				ELSE
					MEMCPY(ADR(strVEVarName),ADR(arrVEOutput)+4+4+4+4+4,SIZEOF(strVEVarName));
				END_IF
												
				IF nVEMaxIndex1 > 0 THEN
					nListIndexArrayStart := nListIndex;
					FOR nVEArrayIndex := 0 TO nVEMaxIndex2-1 DO						
						strVEDisplayVarName := CONCAT(strVEVarName,'[');
						strVEDisplayVarName := CONCAT(strVEDisplayVarName,UDINT_TO_STRING(nVEArrayIndex));
						strVEDisplayVarName := CONCAT(strVEDisplayVarName,']');			
						stCNCVariablesViewer_Data_Temp[nListIndex].strName := strVEDisplayVarName;
						IF (nListIndex < MAX_CNC_VAR_LIST_IDX) THEN
							nListIndex := nListIndex+1;
						ELSE
							EXIT;
						END_IF
							
					END_FOR	
					   nVEArrayIndex := 0;
					   nListIndex := nListIndexArrayStart;
					   nState := 25;											
				ELSE			
					nVEArrayIndex := 0;
					stCNCVariablesViewer_Data_Temp[nListIndex].strName := strVEVarName;						
					nState := 25;
				END_IF						
			END_IF
		END_IF	
		
25:		// Read Value By Name	
		IF nVEMaxIndex1 = 0 THEN			
			strVEVarName := stCNCVariablesViewer_Data_Temp[nListIndex].strName;
		ELSE
			strVEVarName := stCNCVariablesViewer_Data_Temp[nListIndex+nVEArrayIndex].strName ;
		END_IF		
							
		fbReadWrite(
		NETID:= , 
		PORT:= 552, 
		IDXGRP:= 16#22300 + INT_TO_UDINT(nChanIdx)+1, 
		IDXOFFS:= 16#48, 
		WRITELEN:= SIZEOF(strVEVarName), 
		READLEN:= 2048, 
		SRCADDR:= ADR(strVEVarName), 
		DESTADDR:=ADR(arrVEOutput), 
		WRTRD:= TRUE);
		
		IF NOT fbReadWrite.Busy THEN
			IF fbReadWrite.Err	THEN
				Error := fbReadWrite.ERR;
				ErrorID := fbReadWrite.ERRID;
				nState := 99;
			ELSE	
						
				IF nVEType = E_VEVariablesType.BOOLEAN THEN 
					MEMCPY(ADR(dummyBoolean),ADR(arrVEOutput),1);
					strValue := BOOL_TO_STRING(dummyBoolean);
				ELSIF nVEType = E_VEVariablesType.UNS08 THEN
					MEMCPY(ADR(dummyUSInt),ADR(arrVEOutput),1);
					strValue := USINT_TO_STRING(dummyUSInt);
				ELSIF nVEType = E_VEVariablesType.SGN08 THEN
					MEMCPY(ADR(dummySInt),ADR(arrVEOutput),1);
					strValue := SINT_TO_STRING(dummySInt);
				ELSIF nVEType = E_VEVariablesType.UNS16 THEN
					MEMCPY(ADR(dummyUInt),ADR(arrVEOutput),2);
					strValue := UINT_TO_STRING(dummyUInt);
				ELSIF nVEType = E_VEVariablesType.SGN16 THEN
					MEMCPY(ADR(dummyInt),ADR(arrVEOutput),2);
					strValue := INT_TO_STRING(dummyInt);
				ELSIF nVEType = E_VEVariablesType.UNS32 THEN
					MEMCPY(ADR(dummyUDInt),ADR(arrVEOutput),4);
					strValue := UDINT_TO_STRING(dummyUDInt);
				ELSIF nVEType = E_VEVariablesType.SGN32 THEN
					MEMCPY(ADR(dummyDInt),ADR(arrVEOutput),4);
					strValue := DINT_TO_STRING(dummyDInt);
				ELSIF nVEType = E_VEVariablesType.REAL64 THEN
					MEMCPY(ADR(dummyLReal),ADR(arrVEOutput),8);
					strValue := LREAL_TO_STRING(dummyLReal);						
				ELSIF nVEType = E_VEVariablesType.VESTRING THEN					 									
					MEMCPY(ADR(dummyLargeString),ADR(arrVEOutput),nVESize-1);
					strValue := dummyLargeString;
				ELSE
					nState := 99;
				END_IF				
				
				nState := 26;	
			END_IF
		END_IF	
		
26:
		stCNCVariablesViewer_Data_Temp[nListIndex+nVEArrayIndex].strValue := strValue;									
										
		IF nVEArrayIndex < nVEMaxIndex2-1 AND  nVEMaxIndex1 <> 0 THEN
			fbReadWrite(WRTRD:= FALSE);
			nVEArrayIndex := nVEArrayIndex +1;
			IF (nListIndex+nVEArrayIndex <= MAX_CNC_VAR_LIST_IDX) THEN
				nState := 25;
			ELSE
				nState := 60;
			END_IF
		ELSE
			IF (nListIndex <= MAX_CNC_VAR_LIST_IDX) THEN
				nListIndex := nListIndex+nVEArrayIndex +1;
				nState := 30;
			ELSE
				nState := 60;
			END_IF		
			
		END_IF
		
30:  
	IF nIndex < DINT_TO_UDINT(nParameterNumber-1) THEN
		fbReadWrite(WRTRD:= FALSE);		 
		nIndex := nIndex + 1;
		nState := 21;
	ELSE
		fbReadWrite(WRTRD:= FALSE);				
		fbTimer(IN:=FALSE);			
		nState := 60;
	END_IF

60:
	// Output
	Tc2_System.MEMCPY(ADR(stCNCVariablesViewer_Data),ADR(stCNCVariablesViewer_Data_Temp),SIZEOF(stCNCVariablesViewer_Data_Temp));
	fbTimer(IN:=TRUE , PT:=tIntervall);	
	IF fbTimer.Q THEN
		fbReadNumber(READ:= FALSE);
		fbReadWrite(WRTRD:= FALSE);
		nListIndex := 0;
		nIndex := 1;
		nState := 1;
	END_IF

99: // Error 
	nIndex := 1;
	nListIndex := 0;
	fbReadNumber(READ:= FALSE);
	fbReadWrite(WRTRD:= FALSE);
	fbTimer(IN:=FALSE);
	nState := 60;			
END_CASE

END_FUNCTION_BLOCK

// ---- CNC Beckhoff/4 MHT-Function/HLI3_FastMFunctionProvider.TcPOU
FUNCTION_BLOCK HLI3_FastMFunctionProvider
VAR_INPUT
	nHliChanIdx				: UINT;													(* HLI channel index of the channel to check for new M functions *)
	anMFunctionNo			: ARRAY[0..MAX_FAST_M_FUNC_ITEM_IDX] OF UINT;			(* List of M functions munbers to handle *)
END_VAR
VAR_OUTPUT
	stData					: ST_FastMFunctionData;									(* Output structure containing informatione about the handled M functions and their execution offsets *)
	bUnknownChannelIndex	: BOOL;													(* TRUE if the given nHliChanIdx is unknown *)
END_VAR
VAR
	bExitAll				: BOOL;
	bFirstCycle				: BOOL := TRUE;
	byTaskIndex				: BYTE;
	nConfiguredFunctions	: UINT;
	nFunctionCount			: UINT;
	nLoop1					: UINT;
	nLoop2					: UINT;
	anMFunctionNoOld		: ARRAY[0..MAX_FAST_M_FUNC_ITEM_IDX] OF UINT;
	pChan					: POINTER TO HIGH_LEVEL_INTERFACE_CH;
	pData					: POINTER TO ST_FastMFunctionItem;
	pTechno					: POINTER TO Techno_Unit_Ch;
	pMHTechno				: POINTER TO HLI_M_H_Prozess;
	
	fbGetTaskIndex			: Tc2_System.GETCURTASKINDEX;
END_VAR

(****************************************************************************************)
(* POU:		HLI3_FastMFunctionProvider                     								*)
(* Type:	FB																			*)
(* Author: 	RCH		                                             						*)
(* Date: 	14/10/29																	*)
(* Rev.: 	1.0                                               							*)
(* ------------------------------------------------------------------------------------ *)
(* Desc.:	FB for handling CNC M functions contained in the input array				*)
(*			'anMFunctionNo'. These M functions have to be configured as MOS_TS. Their	*)
(*			metadata will be copied into the output structure 'stData' to be processed	*)
(*			by instances of the FB HLI3_FastMFunctionHandler!							*)				
(*																						*)
(*			THIS FB HAS TO BE CALLED CYCLICALLY IN A 1MS TASK!!!						*)
(* ------------------------------------------------------------------------------------ *)
(* Rev.:	1.1																			*)
(* Date:	15/05/05								                                   	*)
(* Author:	RCH																		 	*)
(* Desc.:	Fixed issues occured if more than 1 MOS_TS M function was programmed in a   *)
(*			single G-Code block.														*)
(* ------------------------------------------------------------------------------------ *)
(* Rev.:	<Enter revision number here>												*)
(* Date:	<Enter revision data here>				                                   	*)
(* Author:	<Enter author´s shortcut here>											 	*)
(* Desc.:	<Enter description here>													*)
(****************************************************************************************)

(****************************************************************************************)
(*	  Read current (PLC) task id and check whether the cycle time has been exceeded		*)
(****************************************************************************************)
IF bFirstCycle THEN
	fbGetTaskIndex
		(index				=> byTaskIndex);
END_IF

(****************************************************************************************)
(*								Initialize output structure								*)
(****************************************************************************************)
Tc2_System.MEMSET(ADR(stData), 16#00, SIZEOF(stData));

stData.bCycleTimeExceeded	:= TwinCAT_SystemInfoVarList._TaskInfo[byTaskIndex].CycleTimeExceeded;
stData.bDataValid			:= FALSE;
stData.nFunctionCount		:= 0;	

(****************************************************************************************)
(*	  					  Check existence of the given channel index					*)
(****************************************************************************************)
IF NOT HLI3_CheckChannelValid(nChannel := nHliChanIdx) THEN
	bUnknownChannelIndex	:=	TRUE; 
	RETURN;
ELSE
	bUnknownChannelIndex	:=	FALSE;
END_IF

(****************************************************************************************)
(*	  				  Determine the number of configured M functions					*)
(****************************************************************************************)
IF (Tc2_System.MEMCMP(ADR(anMFunctionNo), ADR(anMFunctionNoOld), SIZEOF(anMFunctionNo)) <> 0) THEN
	anMFunctionNoOld				:= anMFunctionNo;
	nConfiguredFunctions			:= 0;
	
	FOR nLoop1 := 0 TO MAX_FAST_M_FUNC_ITEM_IDX DO
		IF (anMFunctionNoOld[nLoop1] > 0) THEN
			nConfiguredFunctions	:= nConfiguredFunctions + 1;
		END_IF
	END_FOR
END_IF

(****************************************************************************************)
(*	  					  	Check occurances of M functions								*)
(****************************************************************************************)
stData.bDataValid					:= TRUE;
bFirstCycle							:= FALSE;

IF (gpCh[nHliChanIdx]^.used_units_std_sync_r = 0) THEN
	RETURN;
END_IF

pChan								:= gpCh[nHliChanIdx];
nFunctionCount						:= 0;
nLoop1 								:= 0;

FOR nLoop1 := 0 TO INT_TO_UINT(HLI_TU_CH_STD_SYNC_MAXIDX) DO
	IF pChan^.techno_unit_std_sync[nLoop1].please_rw AND (pChan^.techno_unit_std_sync[nLoop1].fkt_ctrl_r = Tc2_CncHli.HLI_INTF_M_FKT) THEN
		pTechno						:= ADR(pChan^.techno_unit_std_sync[nLoop1]);
		pMHTechno					:= ADR(pTechno^.attribut_r);	
		
		(* Check whether this FB has to handle the current M function *)
		FOR nLoop2 := 0 TO (nConfiguredFunctions - 1) DO
			IF (pMHTechno^.nr = anMFunctionNo[nLoop2]) THEN
				pData				:= ADR(stData.astItem[nFunctionCount]);
				pData^.nFunctionNo	:= anMFunctionNo[nLoop2];
				pData^.nOffset		:= pMHTechno^.zeit;
				pData^.nCycleCount	:= TwinCAT_SystemInfoVarList._TaskInfo[byTaskIndex].CycleCount;
				
				nFunctionCount		:= nFunctionCount + 1;
				
				pTechno^.please_rw	:= FALSE;
				pTechno^.done_w		:= TRUE;		
				EXIT;	
			END_IF					
		END_FOR
		
		IF (nFunctionCount >= nConfiguredFunctions) THEN
			EXIT;
		END_IF
	ELSIF NOT pChan^.techno_unit_std_sync[nLoop1].please_rw THEN
		EXIT;
	END_IF	
END_FOR

stData.nFunctionCount				:= nFunctionCount;

END_FUNCTION_BLOCK

// ---- CNC Beckhoff/4 MHT-Function/HLI3_FastMFunctionHandler.TcPOU
FUNCTION_BLOCK HLI3_FastMFunctionHandler
VAR_INPUT
	bForceOff			: BOOL;													(* Forces all bytes in the output array to be 00 and therefore to switch off the digital output *) 
	bReset				: BOOL;													(* Resets the digital output *)
	nFunctionNoOn		: UINT;													(* Specifies the M function number for switching the digital output on *) 
	nDelayOn			: DINT;													(* Specifies a delay time in [µs] for switching on the digital output *)
	nFunctionNoOff		: UINT;													(* Specifies the M function number for switching the digital output off *)
	nDelayOff			: DINT;													(* Specifies a delay time in [µs] for switching off the digital output *)
	stData				: ST_FastMFunctionData;									(* Structure provided by an instance of HLI3_FastMFunctionProvider *)
END_VAR
VAR_OUTPUT
	abyOutput			: ARRAY[0..MAX_FAST_M_FUNC_OUTPUT_IDX] OF BYTE;		(* Output array for a digital oversampling output terminal EL2262 *)  
END_VAR
VAR
	bSwitchOn			: BOOL;
	nSwitchOnOffset		: DINT;
	bSwitchOff			: BOOL;
	nSwitchOffOffset	: DINT;
	bStateChanged		: BOOL;
	bFirstCycle			: BOOL := TRUE;
	byStaticValue		: BYTE;
	byBitmask			: BYTE;
	nBits				: DINT;
	nBytes				: DINT;
	nLoop				: UINT;
	nQueuedCount		: UINT;
	
	eLastState			: E_FastMFunctionState := E_FastMFunctionState.OFF;
	stDequeued			: ST_FastMFunctionBufferItem;
	astQueue			: ARRAY[0..MAX_FAST_M_FUNC_QUEUE_IDX] OF ST_FastMFunctionBufferItem;
	
	fbRtrigReset		: Tc2_Standard.R_TRIG;
	CYCLE_TIME			: UINT := 1000;
END_VAR

(****************************************************************************************)
(* POU:		HLI3_FastMFunctionHandler                     								*)
(* Type:	FB																			*)
(* Author: 	RCH		                                             						*)
(* Date: 	14/10/29																	*)
(* Rev.: 	1.0                                               							*)
(* ------------------------------------------------------------------------------------ *)
(* Desc.:	Function block for handling the oversampled output on an EL2262. The 		*)
(*			output state will be derived from the occurance of two CNC M functions, 	*)
(*			which have to be configured with output method MOS_TS and which have to be	*)
(*			preprocessed by an instance of the HLI3_FastMFunctionProvider function 		*)
(*			block. The switch ON/OFF times can be delayed seperately.					*)					
(*																						*)
(*			THIS FB HAS TO BE CALLED CYCLICALLY IN A 1MS TASK AND THE EL2262 HAS TO 	*)
(*			FEATURE AN OVERSAMPLING FACTOR OF 1000 (125 BYTE) ==> 1µs == 1 bit!!!		*)
(* ------------------------------------------------------------------------------------ *)
(* Rev.:	1.1																			*)
(* Date:	15/05/05								                                   	*)
(* Author:	RCH																		 	*)
(* Desc.:	Fixed issues occured if more than 1 MOS_TS M function was programmed in a   *)
(*			single G-Code block.														*)
(* ------------------------------------------------------------------------------------ *)
(* Rev.:	<Enter revision number here>												*)
(* Date:	<Enter revision data here>				                                   	*)
(* Author:	<Enter author´s shortcut here>											 	*)
(* Desc.:	<Enter description here>													*)
(****************************************************************************************)

(****************************************************************************************)
(*	  						  Refresh buffered switch times 							*)
(****************************************************************************************)
THIS^.RefreshQueue(CYCLE_TIME);

(****************************************************************************************)
(*	  							 	  Reset output										*)
(****************************************************************************************)
fbRtrigReset(CLK:= bReset);

IF fbRtrigReset.Q THEN
	THIS^.ClearQueue();
	bStateChanged				:= TRUE;
	eLastState					:= E_FastMFunctionState.OFF;
END_IF

(****************************************************************************************)
(*	  					    Search for new switch on/off events 						*)
(****************************************************************************************)
bSwitchOn						:= FALSE;
nSwitchOnOffset					:= 0;
bSwitchOff						:= FALSE;
nSwitchOffOffset				:= 0;
nLoop							:= 0;

IF (stData.nFunctionCount > 0) AND (stData.bDataValid) THEN
	REPEAT
		IF (stData.astItem[nLoop].nFunctionNo = nFunctionNoOn) THEN
			bSwitchOn			:= TRUE;
			nSwitchOnOffset		:= stData.astItem[nLoop].nOffset;
		ELSIF (stData.astItem[nLoop].nFunctionNo = nFunctionNoOff) THEN
			bSwitchOff			:= TRUE;
			nSwitchOffOffset	:= stData.astItem[nLoop].nOffset;
		END_IF
	
		nLoop					:= nLoop + 1;
		
		UNTIL ((bSwitchOn AND bSwitchOff) OR (nLoop >= stData.nFunctionCount))
	END_REPEAT	
END_IF

(****************************************************************************************)
(*	  		Buffer found switch on/off events with correspondent switch times			*)
(****************************************************************************************)
IF bSwitchOn AND bSwitchOff THEN
	(* In case switch on and off events have been transmitted within the same cycle, 	*)
	(* order them according to their switch times!										*)
	IF ((nSwitchOnOffset + nDelayOn) < (nSwitchOffOffset + nDelayOff)) THEN
		THIS^.Enqueue(E_FastMFunctionState.ON, nSwitchOnOffset + nDelayOn);
		THIS^.Enqueue(E_FastMFunctionState.OFF, nSwitchOffOffset + nDelayOff); 
	ELSE
		THIS^.Enqueue(E_FastMFunctionState.OFF, nSwitchOffOffset + nDelayOff);
		THIS^.Enqueue(E_FastMFunctionState.ON, nSwitchOnOffset + nDelayOn);
	END_IF
ELSIF bSwitchOn THEN
	THIS^.Enqueue(E_FastMFunctionState.ON, nSwitchOnOffset + nDelayOn);
ELSIF bSwitchOff THEN
	THIS^.Enqueue(E_FastMFunctionState.OFF, nSwitchOffOffset + nDelayOff);
END_IF

(****************************************************************************************)
(*	  				  Set output array according to latest switch state					*)
(****************************************************************************************)
IF bStateChanged OR bFirstCycle THEN
	bStateChanged				:= FALSE;

	IF (eLastState = E_FastMFunctionState.OFF) THEN
		byStaticValue			:= 16#00;
	ELSIF (eLastState = E_FastMFunctionState.ON) THEN
		byStaticValue			:= 16#FF;
	END_IF
	
	Tc2_System.MEMSET(ADR(abyOutput[0]), byStaticValue, SIZEOF(abyOutput));
END_IF

(****************************************************************************************)
(*	  					  Dequeue switch events from the buffer							*)
(****************************************************************************************)
WHILE THIS^.DequeuingRequired DO
	stDequeued					:= THIS^.Dequeue();
	nBits 						:= stDequeued.nSwitchTime MOD 8;
	nBytes 						:= stDequeued.nSwitchTime / 8;
	bStateChanged				:= TRUE;
	IF (stDequeued.nSwitchTime < 0) OR (stDequeued.nSwitchTime > 1000) THEN
		;
	ELSE
		IF ((stDequeued.eState = E_FastMFunctionState.ON) AND (eLastState = E_FastMFunctionState.OFF)) THEN
			byBitmask			:= SHL(BYTE#255, nBits);
			abyOutput[nBytes]	:= abyOutput[nBytes] OR byBitmask;
			eLastState			:= E_FastMFunctionState.ON;
			Tc2_System.MEMSET(ADR(abyOutput[nBytes + 1]), 16#FF, MAX_FAST_M_FUNC_OUTPUT_IDX - nBytes);
		ELSIF ((stDequeued.eState = E_FastMFunctionState.OFF) AND (eLastState = E_FastMFunctionState.ON)) THEN
			byBitmask			:= SHR(BYTE#255, 8 - nBits);
			abyOutput[nBytes]	:= abyOutput[nBytes] AND byBitmask;
			eLastState			:= E_FastMFunctionState.OFF;
			Tc2_System.MEMSET(ADR(abyOutput[nBytes + 1]), 16#00, MAX_FAST_M_FUNC_OUTPUT_IDX - nBytes);
		END_IF
	END_IF
END_WHILE

(****************************************************************************************)
(*	  							   Reset first cycle indicator							*)
(****************************************************************************************)
bFirstCycle						:= FALSE;

PROPERTY DequeuingRequired : BOOL
GET
DequeuingRequired	:= (nQueuedCount > 0) AND 
					   (astQueue[0].eState <> E_FastMFunctionState.EMPTY) AND
					   (astQueue[0].nSwitchTime < CYCLE_TIME);
END_GET
END_PROPERTY

METHOD ClearQueue
Tc2_System.MEMSET(ADR(astQueue), 16#00, SIZEOF(astQueue));
nQueuedCount := 0;
END_METHOD

METHOD Dequeue : ST_FastMFunctionBufferItem
VAR
	stReturn	: ST_FastMFunctionBufferItem;
END_VAR
IF (nQueuedCount > 0) THEN
	stReturn		:=	astQueue[0]; 
	Tc2_System.MEMMOVE(ADR(astQueue[0]), ADR(astQueue[1]), SIZEOF(astQueue) - SIZEOF(stReturn));
	
	nQueuedCount	:= nQueuedCount - 1;
	Dequeue			:= stReturn;
END_IF
END_METHOD

METHOD RefreshQueue
VAR_INPUT
	nCycleTime: UINT;
END_VAR
IF (nQueuedCount > 0) THEN
	FOR nLoop := 0 TO (nQueuedCount - 1) DO
		astQueue[nLoop].nSwitchTime	:= astQueue[nLoop].nSwitchTime - nCycleTime;
	END_FOR
END_IF
END_METHOD

METHOD Enqueue
VAR_INPUT
	eState			: E_FastMFunctionState;
	nSwitchTime		: DINT;
END_VAR
IF (nQueuedCount <= MAX_FAST_M_FUNC_OUTPUT_IDX) THEN
	astQueue[nQueuedCount].eState		:= eState;
	astQueue[nQueuedCount].nSwitchTime	:= nSwitchTime;
	nQueuedCount						:= nQueuedCount + 1;
END_IF
END_METHOD

END_FUNCTION_BLOCK

// ---- CNC Beckhoff/3 Control/FB_Diag.TcPOU
FUNCTION_BLOCK FB_Diag
VAR_OUTPUT
	Alarm: BOOL;
	Vorwarn: BOOL;
	Meld: BOOL;
END_VAR

Alarm := TRUE;
Vorwarn := TRUE;
Meld := TRUE;

END_FUNCTION_BLOCK

// ---- CNC Beckhoff/3 Control/HLI3_ChannelSetEmergencyStop.TcPOU
FUNCTION HLI3_ChannelSetEmergencyStop : BOOL
VAR_INPUT
	/// Number of channel 
	nChanIdx: INT;
	bEStop: BOOL;
END_VAR

(****************************************************************************************)
(* POU:			HLI_ChannelSetEmergenyStop												*)
(* Type:		Function block															*)
(* Customer:	Common																	*)
(* Date:		09/03/12																*)
(* Last:		20/11/12																*)
(* ------------------------------------------------------------------------------------ *)
(* Revision:	1.0																		*)
(* Author:		HR,MiB																	*)
(* Description: (Re-)Sets the channel specific emergency stop unit.						*)
(****************************************************************************************)

HLI3_ChannelSetEmergencyStop := FALSE;
IF NOT HLI3_CheckChannelValid(nChannel := nChanIdx) THEN
	RETURN;
END_IF

(* if the stop button from the HMI is selected the request is set *)
gpCh[nChanIdx]^.bahn_mc_control.emergency_stop.command_w := bEStop;

HLI3_ChannelSetEmergencyStop		:= TRUE;

END_FUNCTION

// ---- CNC Beckhoff/3 Control/HLI3_ChannelSetSuspendAxisOutput.TcPOU
FUNCTION HLI3_ChannelSetSuspendAxisOutput : BOOL
VAR_INPUT
	/// Number of channel 
	nChanIdx: INT;
	bSuspendAxis: BOOL;
END_VAR

(* ========================================================= *)
(*    FUN: HLI_ChannelSuspendAxisOutput                      *)
(* --------------------------------------------------------- *)
(*   Desc:                                                   *)
(* Author: MK , MiB                                          *)
(*   Date: 20.11.2012                                        *)
(*   Rev.: 1.1                                               *)
(* ========================================================= *)
HLI3_ChannelSetSuspendAxisOutput := TRUE;
IF NOT HLI3_CheckChannelValid(nChannel := nChanIdx) THEN
	RETURN;
END_IF
gpCh[nChanIdx]^.bahn_mc_control.suspend_axis_output.command_w := bSuspendAxis;
HLI3_ChannelSetSuspendAxisOutput := TRUE;

END_FUNCTION

// ---- CNC Beckhoff/3 Control/HLI3_ClearReferencePosition.TcPOU
FUNCTION HLI3_ClearReferencePosition : BOOL
VAR_INPUT
	bExecute: BOOL;
	nHliAxisIdx: INT;
END_VAR

(* ========================================================= *)
(*    FUN: HLI3_ClearReferencePosition                       *)
(* --------------------------------------------------------- *)
(*   Desc:                                                   *)
(* 	 Author: TV                                              *)
(*   Date: 17.06.2015                                        *)
(*   Rev.: 1.0                                               *)
(* ========================================================= *)
HLI3_ClearReferencePosition := FALSE;

IF NOT HLI3_CheckAxisValid(nHliAxisIdx := nHliAxisIdx) THEN	
	RETURN;
END_IF

(* set reference position *)
gpAx[nHliAxisIdx]^.lr_mc_control.clear_reference_position.enable_w := TRUE;
gpAx[nHliAxisIdx]^.lr_mc_control.clear_reference_position.command_w := bExecute;
HLI3_ClearReferencePosition := TRUE;

END_FUNCTION

// ---- CNC Beckhoff/3 Control/HLI3_GetActualAxisPos.TcPOU
FUNCTION HLI3_GetActualAxisPos : LREAL
VAR_INPUT
	///Achs ID
	nHliAxisIdx: INT;
END_VAR
VAR
	HLI_GetActualAxisPos: DINT;
END_VAR



IF NOT (HLI3_CheckAxisValid(nHliAxisIdx := nHliAxisIdx)) THEN
	HLI3_GetActualAxisPos := -1;
	RETURN;
END_IF

HLI3_GetActualAxisPos:=  gpAx[nHliAxisIdx]^.lr_state.current_position_acs_r;

END_FUNCTION

// ---- CNC Beckhoff/3 Control/HLI3_GetAxisReferenceState.TcPOU
FUNCTION HLI3_GetAxisReferenceState : BOOL
VAR_INPUT
	nHliAxisIdx: INT;
END_VAR


IF NOT HLI3_CheckAxisValid(nHliAxisIdx := nHliAxisIdx) THEN
	HLI3_GetAxisReferenceState := FALSE;
	RETURN;
END_IF

HLI3_GetAxisReferenceState:= gpAx[nHliAxisIdx]^.lr_state.homing_done_r;

END_FUNCTION

